KUKA KRL program: PPR_fullpath_2mm_split2.src

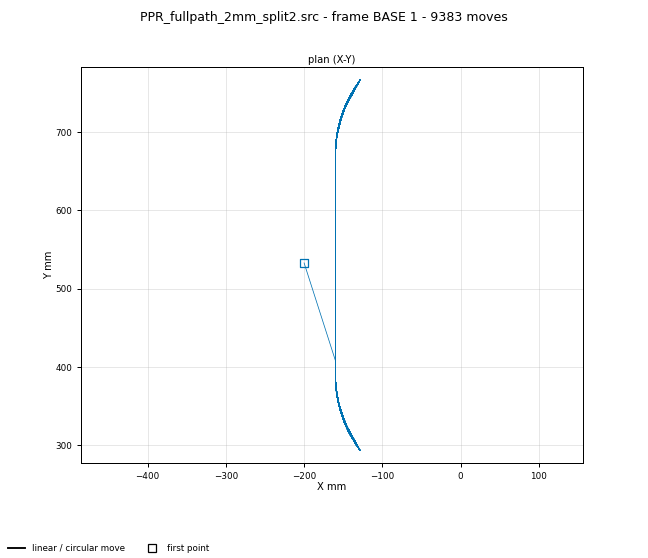
[picture p0: tool path of PPR_fullpath_2mm_split2.src in frame BASE 1, 9383 of 9384 moves have a stored position in this frame; points joined in program order, loops and branches not executed]
&ACCESS RVEO
&REL 11
&PARAM TEMPLATE = C:\KRC\Roboter\Template\vorgabe
&PARAM EDITMASK = *
DEF variable_helical2( )
;FOLD INI
  ;FOLD BASISTECH INI
    GLOBAL INTERRUPT DECL 3 WHEN $STOPMESS==TRUE DO IR_STOPM ( )
    INTERRUPT ON 3
    BAS (#INITMOV,0 )
  ;ENDFOLD (BASISTECH INI)
 ;FOLD USER INI


    ;Make your modifications here
  ;ENDFOLD (USER INI)
;ENDFOLD (INI)
ACTION(#AXIS_RESET,34,1000,#NOERROR,ERROR_CODE)
;FOLD PTP HOME  Vel= 100 % DEFAULT;%{PE}%MKUKATPBASIS,%CMOVE,%VPTP,%P 1:PTP, 2:HOME, 3:, 5:100, 7:DEFAULT
$BWDSTART = FALSE
PDAT_ACT=PDEFAULT
FDAT_ACT=FHOME
BAS (#PTP_PARAMS,100 )
$H_POS=XHOME
PTP  XHOME
;ENDFOLD
BAS(#TOOL,1)
BAS(#BASE,1)
$VEL_AXIS[1]=100
$VEL_AXIS[2]=100
$VEL_AXIS[3]=100
$VEL_AXIS[4]=100
$VEL_AXIS[5]=100
$VEL_AXIS[6]=100
$VEL_EXTAX[1]=100
$VEL_EXTAX[2]=100

$ACC_AXIS[1]=100
$ACC_AXIS[2]=100
$ACC_AXIS[3]=100
$ACC_AXIS[4]=100
$ACC_AXIS[5]=100
$ACC_AXIS[6]=100
$ACC_EXTAX[1]=100
$ACC_EXTAX[2]=100

SLIN {X  -200.000, Y  +533.000, Z    +0.000, A    +0.000, E1    +0.000, E3    +0.000, E4    +0.000}

SLIN {X  -160.000, Y  +408.284, Z    +0.000, E1   +56.435, E3  -372.434}
HALT
SPLINE
SPL {X  -160.000, Y  +395.668, Z    +0.000, E1   +56.446, E3  -354.661}
SPL {X  -159.894, Y  +382.991, Z    +0.000, E1   +56.419, E3  -336.663}
SPL {X  -159.213, Y  +372.948, Z    +0.000, E1   +56.290, E3  -321.768}
SPL {X  -158.141, Y  +364.480, Z    +0.000, E1   +56.110, E3  -308.694}
SPL {X  -156.499, Y  +355.511, Z    +0.000, E1   +55.854, E3  -294.378}
SPL {X  -154.489, Y  +347.168, Z    +0.000, E1   +55.487, E3  -280.503}
SPL {X  -152.108, Y  +339.170, Z    +0.000, E1   +55.085, E3  -266.814}
SPL {X  -149.149, Y  +330.880, Z    +0.000, E1   +54.560, E3  -252.178}
SPL {X  -146.188, Y  +323.769, Z    +0.000, E1   +53.991, E3  -239.222}
SPL {X  -143.516, Y  +318.068, Z    +0.000, E1   +53.476, E3  -228.622}
SPL {X  -140.415, Y  +312.095, Z    +0.000, E1   +52.896, E3  -217.355}
SPL {X  -128.706, Y  +293.749, Z    +0.000, E1   +44.636, E3  -115.294}
ENDSPLINE

SPLINE
SPL {X  -149.341, Y  +331.377, Z    +0.000, E1   +30.257, E3   -35.419}
SPL {X  -155.855, Y  +352.616, Z    +0.000, E1   +20.935, E3   -23.306}
SPL {X  -158.820, Y  +369.405, Z    +0.000, E1   +11.982, E3   -17.902}
SPL {X  -159.764, Y  +380.110, Z    +0.000, E1    +5.506, E3   -16.035}
SPL {X  -159.978, Y  +386.129, Z    +0.000, E1    +1.351, E3   -15.453}
SPL {X  -160.000, Y  +390.626, Z    +0.000, E1    -2.404, E3   -15.189}
SPL {X  -160.000, Y  +397.252, Z    +0.000, E1   -10.844, E3   -14.488}
SPL {X  -160.000, Y  +404.580, Z    +0.000, E1   -20.626, E3   -13.063}
SPL {X  -160.000, Y  +414.518, Z    +0.000, E1   -32.156, E3    -9.972}
SPL {X  -160.000, Y  +450.190, Z    +0.000, E1   -50.789, E3   +10.114}
SPL {X  -160.000, Y  +522.988, Z    +0.000, E1   -55.744, E3   +88.448}
SPL {X  -160.000, Y  +538.972, Z    +0.000, E1   -55.709, E3  +111.680}
SPL {X  -160.000, Y  +554.704, Z    +0.000, E1   -55.732, E3  +134.447}
SPL {X  -160.000, Y  +570.552, Z    +0.000, E1   -55.716, E3  +157.461}
SPL {X  -160.000, Y  +586.464, Z    +0.000, E1   -55.733, E3  +180.507}
SPL {X  -160.000, Y  +602.947, Z    +0.000, E1   -55.730, E3  +204.403}
SPL {X  -160.000, Y  +618.907, Z    +0.000, E1   -55.724, E3  +227.541}
SPL {X  -160.000, Y  +633.674, Z    +0.000, E1   -55.717, E3  +248.961}
SPL {X  -160.000, Y  +646.135, Z    +0.000, E1   -55.674, E3  +267.102}
SPL {X  -160.000, Y  +658.587, Z    +0.000, E1   -55.708, E3  +285.098}
SPL {X  -160.000, Y  +671.750, Z    +0.000, E1   -55.695, E3  +304.182}
SPL {X  -159.611, Y  +682.650, Z    +0.000, E1   -55.614, E3  +320.420}
SPL {X  -158.677, Y  +692.037, Z    +0.000, E1   -55.461, E3  +335.003}
SPL {X  -157.091, Y  +701.873, Z    +0.000, E1   -55.210, E3  +350.889}
SPL {X  -154.891, Y  +711.608, Z    +0.000, E1   -54.831, E3  +367.276}
SPL {X  -152.273, Y  +720.623, Z    +0.000, E1   -54.369, E3  +383.014}
SPL {X  -149.300, Y  +729.027, Z    +0.000, E1   -53.836, E3  +398.150}
SPL {X  -146.549, Y  +735.713, Z    +0.000, E1   -53.293, E3  +410.565}
SPL {X  -144.128, Y  +740.978, Z    +0.000, E1   -52.835, E3  +420.527}
SPL {X  -141.140, Y  +746.862, Z    +0.000, E1   -52.272, E3  +431.815}
SPL {X  -128.473, Y  +766.865, Z    +0.000, E1   -45.208, E3  +526.024}
ENDSPLINE

SPLINE
SPL {X  -149.609, Y  +728.220, Z    +0.000, E1   -30.103, E3  +611.717}
SPL {X  -157.346, Y  +700.520, Z    +0.000, E1   -17.449, E3  +626.438}
SPL {X  -159.391, Y  +685.442, Z    +0.000, E1    -8.940, E3  +630.323}
SPL {X  -159.974, Y  +674.384, Z    +0.000, E1    -1.914, E3  +631.675}
SPL {X  -160.000, Y  +668.854, Z    +0.000, E1    +3.008, E3  +632.026}
SPL {X  -160.000, Y  +662.175, Z    +0.000, E1   +11.518, E3  +632.797}
SPL {X  -160.000, Y  +654.447, Z    +0.000, E1   +21.734, E3  +634.422}
SPL {X  -160.000, Y  +641.600, Z    +0.000, E1   +35.681, E3  +638.687}
SPL {X  -160.000, Y  +601.361, Z    +0.000, E1   +52.744, E3  +662.649}
SPL {X  -160.000, Y  +531.662, Z    +0.000, E1   +56.951, E3  +734.638}
SPL {X  -160.000, Y  +513.172, Z    +0.000, E1   +56.969, E3  +760.194}
SPL {X  -160.000, Y  +498.160, Z    +0.000, E1   +56.531, E3  +783.807}
ENDSPLINE

SPLINE
SPL {X  -160.000, Y  +512.094, Z    +0.000, E1   +49.085, E3  +807.795}
ENDSPLINE

SPLINE
SPL {X  -160.000, Y  +491.347, Z    +0.000, E1   +50.960, E3  +833.461}
SPL {X  -160.000, Y  +470.538, Z    +0.000, E1   +52.629, E3  +858.147}
SPL {X  -160.000, Y  +453.213, Z    +0.000, E1   +53.894, E3  +877.585}
SPL {X  -160.000, Y  +440.734, Z    +0.000, E1   +54.729, E3  +891.367}
SPL {X  -160.000, Y  +423.596, Z    +0.000, E1   +55.911, E3  +909.259}
SPL {X  -160.000, Y  +408.178, Z    +0.000, E1   +56.432, E3  +927.720}
SPL {X  -160.000, Y  +395.668, Z    +0.000, E1   +56.446, E3  +945.336}
SPL {X  -159.894, Y  +382.991, Z    +0.000, E1   +56.419, E3  +963.334}
SPL {X  -159.213, Y  +372.948, Z    +0.000, E1   +56.290, E3  +978.228}
SPL {X  -158.141, Y  +364.480, Z    +0.000, E1   +56.110, E3  +991.303}
SPL {X  -156.499, Y  +355.511, Z    +0.000, E1   +55.854, E3 +1005.619}
SPL {X  -154.489, Y  +347.168, Z    +0.000, E1   +55.487, E3 +1019.493}
SPL {X  -152.108, Y  +339.170, Z    +0.000, E1   +55.085, E3 +1033.182}
SPL {X  -149.149, Y  +330.880, Z    +0.000, E1   +54.560, E3 +1047.818}
SPL {X  -146.188, Y  +323.769, Z    +0.000, E1   +53.991, E3 +1060.775}
SPL {X  -143.516, Y  +318.068, Z    +0.000, E1   +53.476, E3 +1071.374}
SPL {X  -140.415, Y  +312.095, Z    +0.000, E1   +52.896, E3 +1082.642}
SPL {X  -128.706, Y  +293.749, Z    +0.000, E1   +44.636, E3 +1184.702}
ENDSPLINE

SPLINE
SPL {X  -149.341, Y  +331.377, Z    +0.000, E1   +30.257, E3 +1264.578}
SPL {X  -155.855, Y  +352.616, Z    +0.000, E1   +20.935, E3 +1276.691}
SPL {X  -158.820, Y  +369.405, Z    +0.000, E1   +11.982, E3 +1282.094}
SPL {X  -159.764, Y  +380.110, Z    +0.000, E1    +5.506, E3 +1283.961}
SPL {X  -159.978, Y  +386.129, Z    +0.000, E1    +1.351, E3 +1284.543}
SPL {X  -160.000, Y  +390.626, Z    +0.000, E1    -2.404, E3 +1284.807}
SPL {X  -160.000, Y  +397.252, Z    +0.000, E1   -10.844, E3 +1285.508}
SPL {X  -160.000, Y  +404.580, Z    +0.000, E1   -20.626, E3 +1286.934}
SPL {X  -160.000, Y  +414.518, Z    +0.000, E1   -32.156, E3 +1290.024}
SPL {X  -160.000, Y  +450.190, Z    +0.000, E1   -50.789, E3 +1310.110}
SPL {X  -160.000, Y  +522.988, Z    +0.000, E1   -55.744, E3 +1388.444}
SPL {X  -160.000, Y  +538.972, Z    +0.000, E1   -55.709, E3 +1411.677}
SPL {X  -160.000, Y  +554.704, Z    +0.000, E1   -55.732, E3 +1434.443}
SPL {X  -160.000, Y  +570.552, Z    +0.000, E1   -55.716, E3 +1457.458}
SPL {X  -160.000, Y  +586.464, Z    +0.000, E1   -55.733, E3 +1480.503}
SPL {X  -160.000, Y  +602.947, Z    +0.000, E1   -55.730, E3 +1504.400}
SPL {X  -160.000, Y  +618.907, Z    +0.000, E1   -55.724, E3 +1527.537}
SPL {X  -160.000, Y  +633.674, Z    +0.000, E1   -55.717, E3 +1548.957}
SPL {X  -160.000, Y  +646.135, Z    +0.000, E1   -55.674, E3 +1567.098}
SPL {X  -160.000, Y  +658.587, Z    +0.000, E1   -55.708, E3 +1585.094}
SPL {X  -160.000, Y  +671.750, Z    +0.000, E1   -55.695, E3 +1604.179}
SPL {X  -159.611, Y  +682.650, Z    +0.000, E1   -55.614, E3 +1620.417}
SPL {X  -158.677, Y  +692.037, Z    +0.000, E1   -55.461, E3 +1635.000}
SPL {X  -157.091, Y  +701.873, Z    +0.000, E1   -55.210, E3 +1650.886}
SPL {X  -154.891, Y  +711.608, Z    +0.000, E1   -54.831, E3 +1667.273}
SPL {X  -152.273, Y  +720.623, Z    +0.000, E1   -54.369, E3 +1683.010}
SPL {X  -149.300, Y  +729.027, Z    +0.000, E1   -53.836, E3 +1698.146}
SPL {X  -146.549, Y  +735.713, Z    +0.000, E1   -53.293, E3 +1710.561}
SPL {X  -144.128, Y  +740.978, Z    +0.000, E1   -52.835, E3 +1720.524}
SPL {X  -141.140, Y  +746.862, Z    +0.000, E1   -52.272, E3 +1731.811}
SPL {X  -128.473, Y  +766.865, Z    +0.000, E1   -45.208, E3 +1826.021}
ENDSPLINE

SPLINE
SPL {X  -149.609, Y  +728.220, Z    +0.000, E1   -30.103, E3 +1911.713}
SPL {X  -157.346, Y  +700.520, Z    +0.000, E1   -17.449, E3 +1926.434}
SPL {X  -159.391, Y  +685.442, Z    +0.000, E1    -8.940, E3 +1930.319}
SPL {X  -159.974, Y  +674.384, Z    +0.000, E1    -1.914, E3 +1931.671}
SPL {X  -160.000, Y  +668.854, Z    +0.000, E1    +3.008, E3 +1932.022}
SPL {X  -160.000, Y  +662.175, Z    +0.000, E1   +11.518, E3 +1932.793}
SPL {X  -160.000, Y  +654.447, Z    +0.000, E1   +21.734, E3 +1934.419}
SPL {X  -160.000, Y  +641.600, Z    +0.000, E1   +35.681, E3 +1938.684}
SPL {X  -160.000, Y  +601.361, Z    +0.000, E1   +52.744, E3 +1962.645}
SPL {X  -160.000, Y  +531.662, Z    +0.000, E1   +56.951, E3 +2034.635}
SPL {X  -160.000, Y  +513.172, Z    +0.000, E1   +56.969, E3 +2060.190}
SPL {X  -160.000, Y  +498.160, Z    +0.000, E1   +56.531, E3 +2083.803}
ENDSPLINE

SPLINE
SPL {X  -160.000, Y  +512.094, Z    +0.000, E1   +49.085, E3 +2107.791}
ENDSPLINE

SPLINE
SPL {X  -160.000, Y  +491.347, Z    +0.000, E1   +50.960, E3 +2133.458}
SPL {X  -160.000, Y  +470.538, Z    +0.000, E1   +52.629, E3 +2158.144}
SPL {X  -160.000, Y  +453.213, Z    +0.000, E1   +53.894, E3 +2177.582}
SPL {X  -160.000, Y  +440.734, Z    +0.000, E1   +54.729, E3 +2191.364}
SPL {X  -160.000, Y  +423.596, Z    +0.000, E1   +55.911, E3 +2209.256}
SPL {X  -160.000, Y  +408.178, Z    +0.000, E1   +56.432, E3 +2227.717}
SPL {X  -160.000, Y  +395.668, Z    +0.000, E1   +56.446, E3 +2245.332}
SPL {X  -159.894, Y  +382.991, Z    +0.000, E1   +56.419, E3 +2263.330}
SPL {X  -159.213, Y  +372.948, Z    +0.000, E1   +56.290, E3 +2278.225}
SPL {X  -158.141, Y  +364.480, Z    +0.000, E1   +56.110, E3 +2291.299}
SPL {X  -156.499, Y  +355.511, Z    +0.000, E1   +55.854, E3 +2305.615}
SPL {X  -154.489, Y  +347.168, Z    +0.000, E1   +55.487, E3 +2319.490}
SPL {X  -152.108, Y  +339.170, Z    +0.000, E1   +55.085, E3 +2333.179}
SPL {X  -149.149, Y  +330.880, Z    +0.000, E1   +54.560, E3 +2347.814}
SPL {X  -146.188, Y  +323.769, Z    +0.000, E1   +53.991, E3 +2360.771}
SPL {X  -143.516, Y  +318.068, Z    +0.000, E1   +53.476, E3 +2371.371}
SPL {X  -140.415, Y  +312.095, Z    +0.000, E1   +52.896, E3 +2382.638}
SPL {X  -128.706, Y  +293.749, Z    +0.000, E1   +44.636, E3 +2484.699}
ENDSPLINE

SPLINE
SPL {X  -149.341, Y  +331.377, Z    +0.000, E1   +30.257, E3 +2564.574}
SPL {X  -155.855, Y  +352.616, Z    +0.000, E1   +20.935, E3 +2576.687}
SPL {X  -158.820, Y  +369.405, Z    +0.000, E1   +11.982, E3 +2582.091}
SPL {X  -159.764, Y  +380.110, Z    +0.000, E1    +5.506, E3 +2583.957}
SPL {X  -159.978, Y  +386.129, Z    +0.000, E1    +1.351, E3 +2584.540}
SPL {X  -160.000, Y  +390.626, Z    +0.000, E1    -2.404, E3 +2584.804}
SPL {X  -160.000, Y  +397.252, Z    +0.000, E1   -10.844, E3 +2585.504}
SPL {X  -160.000, Y  +404.580, Z    +0.000, E1   -20.626, E3 +2586.930}
SPL {X  -160.000, Y  +414.518, Z    +0.000, E1   -32.156, E3 +2590.021}
SPL {X  -160.000, Y  +450.190, Z    +0.000, E1   -50.789, E3 +2610.106}
SPL {X  -160.000, Y  +522.988, Z    +0.000, E1   -55.744, E3 +2688.441}
SPL {X  -160.000, Y  +538.972, Z    +0.000, E1   -55.709, E3 +2711.673}
SPL {X  -160.000, Y  +554.704, Z    +0.000, E1   -55.732, E3 +2734.439}
SPL {X  -160.000, Y  +570.552, Z    +0.000, E1   -55.716, E3 +2757.454}
SPL {X  -160.000, Y  +586.464, Z    +0.000, E1   -55.733, E3 +2780.499}
SPL {X  -160.000, Y  +602.947, Z    +0.000, E1   -55.730, E3 +2804.396}
SPL {X  -160.000, Y  +618.907, Z    +0.000, E1   -55.724, E3 +2827.534}
SPL {X  -160.000, Y  +633.674, Z    +0.000, E1   -55.717, E3 +2848.954}
SPL {X  -160.000, Y  +646.135, Z    +0.000, E1   -55.674, E3 +2867.094}
SPL {X  -160.000, Y  +658.587, Z    +0.000, E1   -55.708, E3 +2885.090}
SPL {X  -160.000, Y  +671.750, Z    +0.000, E1   -55.695, E3 +2904.175}
SPL {X  -159.611, Y  +682.650, Z    +0.000, E1   -55.614, E3 +2920.413}
SPL {X  -158.677, Y  +692.037, Z    +0.000, E1   -55.461, E3 +2934.996}
SPL {X  -157.091, Y  +701.873, Z    +0.000, E1   -55.210, E3 +2950.882}
SPL {X  -154.891, Y  +711.608, Z    +0.000, E1   -54.831, E3 +2967.269}
SPL {X  -152.273, Y  +720.623, Z    +0.000, E1   -54.369, E3 +2983.007}
SPL {X  -149.300, Y  +729.027, Z    +0.000, E1   -53.836, E3 +2998.143}
SPL {X  -146.549, Y  +735.713, Z    +0.000, E1   -53.293, E3 +3010.557}
SPL {X  -144.128, Y  +740.978, Z    +0.000, E1   -52.835, E3 +3020.520}
SPL {X  -141.140, Y  +746.862, Z    +0.000, E1   -52.272, E3 +3031.808}
SPL {X  -128.473, Y  +766.865, Z    +0.000, E1   -45.208, E3 +3126.017}
ENDSPLINE

SPLINE
SPL {X  -149.609, Y  +728.220, Z    +0.000, E1   -30.103, E3 +3211.710}
SPL {X  -157.346, Y  +700.520, Z    +0.000, E1   -17.449, E3 +3226.431}
SPL {X  -159.391, Y  +685.442, Z    +0.000, E1    -8.940, E3 +3230.316}
SPL {X  -159.974, Y  +674.384, Z    +0.000, E1    -1.914, E3 +3231.668}
SPL {X  -160.000, Y  +668.854, Z    +0.000, E1    +3.008, E3 +3232.019}
SPL {X  -160.000, Y  +662.175, Z    +0.000, E1   +11.518, E3 +3232.789}
SPL {X  -160.000, Y  +654.447, Z    +0.000, E1   +21.734, E3 +3234.415}
SPL {X  -160.000, Y  +641.600, Z    +0.000, E1   +35.681, E3 +3238.680}
SPL {X  -160.000, Y  +601.361, Z    +0.000, E1   +52.744, E3 +3262.642}
SPL {X  -160.000, Y  +531.662, Z    +0.000, E1   +56.951, E3 +3334.631}
SPL {X  -160.000, Y  +513.172, Z    +0.000, E1   +56.969, E3 +3360.187}
SPL {X  -160.000, Y  +498.160, Z    +0.000, E1   +56.531, E3 +3383.800}
ENDSPLINE

SPLINE
SPL {X  -160.000, Y  +512.094, Z    +0.000, E1   +49.085, E3 +3407.787}
ENDSPLINE

SPLINE
SPL {X  -160.000, Y  +491.347, Z    +0.000, E1   +50.960, E3 +3433.454}
SPL {X  -160.000, Y  +470.538, Z    +0.000, E1   +52.629, E3 +3458.140}
SPL {X  -160.000, Y  +453.213, Z    +0.000, E1   +53.894, E3 +3477.578}
SPL {X  -160.000, Y  +440.734, Z    +0.000, E1   +54.729, E3 +3491.360}
SPL {X  -160.000, Y  +423.596, Z    +0.000, E1   +55.911, E3 +3509.252}
SPL {X  -160.000, Y  +408.178, Z    +0.000, E1   +56.432, E3 +3527.713}
SPL {X  -160.000, Y  +395.668, Z    +0.000, E1   +56.446, E3 +3545.328}
SPL {X  -159.894, Y  +382.991, Z    +0.000, E1   +56.419, E3 +3563.326}
SPL {X  -159.213, Y  +372.948, Z    +0.000, E1   +56.290, E3 +3578.221}
SPL {X  -158.141, Y  +364.480, Z    +0.000, E1   +56.110, E3 +3591.295}
SPL {X  -156.499, Y  +355.511, Z    +0.000, E1   +55.854, E3 +3605.611}
SPL {X  -154.489, Y  +347.168, Z    +0.000, E1   +55.487, E3 +3619.486}
SPL {X  -152.108, Y  +339.170, Z    +0.000, E1   +55.085, E3 +3633.175}
SPL {X  -149.149, Y  +330.880, Z    +0.000, E1   +54.560, E3 +3647.811}
SPL {X  -146.188, Y  +323.769, Z    +0.000, E1   +53.991, E3 +3660.767}
SPL {X  -143.516, Y  +318.068, Z    +0.000, E1   +53.476, E3 +3671.367}
SPL {X  -140.415, Y  +312.095, Z    +0.000, E1   +52.896, E3 +3682.634}
SPL {X  -128.706, Y  +293.749, Z    +0.000, E1   +44.636, E3 +3784.695}
ENDSPLINE

SPLINE
SPL {X  -149.341, Y  +331.377, Z    +0.000, E1   +30.257, E3 +3864.571}
SPL {X  -155.855, Y  +352.616, Z    +0.000, E1   +20.935, E3 +3876.683}
SPL {X  -158.820, Y  +369.405, Z    +0.000, E1   +11.982, E3 +3882.087}
SPL {X  -159.764, Y  +380.110, Z    +0.000, E1    +5.506, E3 +3883.954}
SPL {X  -159.978, Y  +386.129, Z    +0.000, E1    +1.351, E3 +3884.536}
SPL {X  -160.000, Y  +390.626, Z    +0.000, E1    -2.404, E3 +3884.800}
SPL {X  -160.000, Y  +397.252, Z    +0.000, E1   -10.844, E3 +3885.501}
SPL {X  -160.000, Y  +404.580, Z    +0.000, E1   -20.626, E3 +3886.926}
SPL {X  -160.000, Y  +414.518, Z    +0.000, E1   -32.156, E3 +3890.017}
SPL {X  -160.000, Y  +450.190, Z    +0.000, E1   -50.789, E3 +3910.103}
SPL {X  -160.000, Y  +522.988, Z    +0.000, E1   -55.744, E3 +3988.437}
SPL {X  -160.000, Y  +538.972, Z    +0.000, E1   -55.709, E3 +4011.669}
SPL {X  -160.000, Y  +554.704, Z    +0.000, E1   -55.732, E3 +4034.436}
SPL {X  -160.000, Y  +570.552, Z    +0.000, E1   -55.716, E3 +4057.450}
SPL {X  -160.000, Y  +586.464, Z    +0.000, E1   -55.733, E3 +4080.496}
SPL {X  -160.000, Y  +602.947, Z    +0.000, E1   -55.730, E3 +4104.392}
SPL {X  -160.000, Y  +618.907, Z    +0.000, E1   -55.724, E3 +4127.530}
SPL {X  -160.000, Y  +633.674, Z    +0.000, E1   -55.717, E3 +4148.950}
SPL {X  -160.000, Y  +646.135, Z    +0.000, E1   -55.674, E3 +4167.091}
SPL {X  -160.000, Y  +658.587, Z    +0.000, E1   -55.708, E3 +4185.087}
SPL {X  -160.000, Y  +671.750, Z    +0.000, E1   -55.695, E3 +4204.172}
SPL {X  -159.611, Y  +682.650, Z    +0.000, E1   -55.614, E3 +4220.409}
SPL {X  -158.677, Y  +692.037, Z    +0.000, E1   -55.461, E3 +4234.992}
SPL {X  -157.091, Y  +701.873, Z    +0.000, E1   -55.210, E3 +4250.879}
SPL {X  -154.891, Y  +711.608, Z    +0.000, E1   -54.831, E3 +4267.265}
SPL {X  -152.273, Y  +720.623, Z    +0.000, E1   -54.369, E3 +4283.003}
SPL {X  -149.300, Y  +729.027, Z    +0.000, E1   -53.836, E3 +4298.139}
SPL {X  -146.549, Y  +735.713, Z    +0.000, E1   -53.293, E3 +4310.554}
SPL {X  -144.128, Y  +740.978, Z    +0.000, E1   -52.835, E3 +4320.516}
SPL {X  -141.140, Y  +746.862, Z    +0.000, E1   -52.272, E3 +4331.804}
SPL {X  -128.473, Y  +766.865, Z    +0.000, E1   -45.208, E3 +4426.013}
ENDSPLINE

SPLINE
SPL {X  -149.609, Y  +728.220, Z    +0.000, E1   -30.103, E3 +4511.706}
SPL {X  -157.346, Y  +700.520, Z    +0.000, E1   -17.449, E3 +4526.427}
SPL {X  -159.391, Y  +685.442, Z    +0.000, E1    -8.940, E3 +4530.312}
SPL {X  -159.974, Y  +674.384, Z    +0.000, E1    -1.914, E3 +4531.664}
SPL {X  -160.000, Y  +668.854, Z    +0.000, E1    +3.008, E3 +4532.015}
SPL {X  -160.000, Y  +662.175, Z    +0.000, E1   +11.518, E3 +4532.786}
SPL {X  -160.000, Y  +654.447, Z    +0.000, E1   +21.734, E3 +4534.411}
SPL {X  -160.000, Y  +641.600, Z    +0.000, E1   +35.681, E3 +4538.676}
SPL {X  -160.000, Y  +601.361, Z    +0.000, E1   +52.744, E3 +4562.638}
SPL {X  -160.000, Y  +531.662, Z    +0.000, E1   +56.951, E3 +4634.627}
SPL {X  -160.000, Y  +513.172, Z    +0.000, E1   +56.969, E3 +4660.183}
SPL {X  -160.000, Y  +498.160, Z    +0.000, E1   +56.531, E3 +4683.796}
ENDSPLINE

SPLINE
SPL {X  -160.000, Y  +512.094, Z    +0.000, E1   +49.085, E3 +4707.784}
ENDSPLINE

SPLINE
SPL {X  -160.000, Y  +491.347, Z    +0.000, E1   +50.960, E3 +4733.450}
SPL {X  -160.000, Y  +470.538, Z    +0.000, E1   +52.629, E3 +4758.136}
SPL {X  -160.000, Y  +453.213, Z    +0.000, E1   +53.894, E3 +4777.574}
SPL {X  -160.000, Y  +440.734, Z    +0.000, E1   +54.729, E3 +4791.356}
SPL {X  -160.000, Y  +423.596, Z    +0.000, E1   +55.911, E3 +4809.248}
SPL {X  -160.000, Y  +408.178, Z    +0.000, E1   +56.432, E3 +4827.709}
SPL {X  -160.000, Y  +395.668, Z    +0.000, E1   +56.446, E3 +4845.325}
SPL {X  -159.894, Y  +382.991, Z    +0.000, E1   +56.419, E3 +4863.323}
SPL {X  -159.213, Y  +372.948, Z    +0.000, E1   +56.290, E3 +4878.217}
SPL {X  -158.141, Y  +364.480, Z    +0.000, E1   +56.110, E3 +4891.292}
SPL {X  -156.499, Y  +355.511, Z    +0.000, E1   +55.854, E3 +4905.608}
SPL {X  -154.489, Y  +347.168, Z    +0.000, E1   +55.487, E3 +4919.482}
SPL {X  -152.108, Y  +339.170, Z    +0.000, E1   +55.085, E3 +4933.172}
SPL {X  -149.149, Y  +330.880, Z    +0.000, E1   +54.560, E3 +4947.807}
SPL {X  -146.188, Y  +323.769, Z    +0.000, E1   +53.991, E3 +4960.764}
SPL {X  -143.516, Y  +318.068, Z    +0.000, E1   +53.476, E3 +4971.363}
SPL {X  -140.415, Y  +312.095, Z    +0.000, E1   +52.896, E3 +4982.631}
SPL {X  -128.706, Y  +293.749, Z    +0.000, E1   +44.636, E3 +5084.691}
ENDSPLINE

SPLINE
SPL {X  -149.341, Y  +331.377, Z    +0.000, E1   +30.257, E3 +5164.567}
SPL {X  -155.855, Y  +352.616, Z    +0.000, E1   +20.935, E3 +5176.680}
SPL {X  -158.820, Y  +369.405, Z    +0.000, E1   +11.982, E3 +5182.084}
SPL {X  -159.764, Y  +380.110, Z    +0.000, E1    +5.506, E3 +5183.950}
SPL {X  -159.978, Y  +386.129, Z    +0.000, E1    +1.351, E3 +5184.532}
SPL {X  -160.000, Y  +390.626, Z    +0.000, E1    -2.404, E3 +5184.796}
SPL {X  -160.000, Y  +397.252, Z    +0.000, E1   -10.844, E3 +5185.497}
SPL {X  -160.000, Y  +404.580, Z    +0.000, E1   -20.626, E3 +5186.923}
SPL {X  -160.000, Y  +414.518, Z    +0.000, E1   -32.156, E3 +5190.013}
SPL {X  -160.000, Y  +450.190, Z    +0.000, E1   -50.789, E3 +5210.099}
SPL {X  -160.000, Y  +522.988, Z    +0.000, E1   -55.744, E3 +5288.433}
SPL {X  -160.000, Y  +538.972, Z    +0.000, E1   -55.709, E3 +5311.666}
SPL {X  -160.000, Y  +554.704, Z    +0.000, E1   -55.732, E3 +5334.432}
SPL {X  -160.000, Y  +570.552, Z    +0.000, E1   -55.716, E3 +5357.447}
SPL {X  -160.000, Y  +586.464, Z    +0.000, E1   -55.733, E3 +5380.492}
SPL {X  -160.000, Y  +602.947, Z    +0.000, E1   -55.730, E3 +5404.389}
SPL {X  -160.000, Y  +618.907, Z    +0.000, E1   -55.724, E3 +5427.527}
SPL {X  -160.000, Y  +633.674, Z    +0.000, E1   -55.717, E3 +5448.947}
SPL {X  -160.000, Y  +646.135, Z    +0.000, E1   -55.674, E3 +5467.087}
SPL {X  -160.000, Y  +658.587, Z    +0.000, E1   -55.708, E3 +5485.083}
SPL {X  -160.000, Y  +671.750, Z    +0.000, E1   -55.695, E3 +5504.168}
SPL {X  -159.611, Y  +682.650, Z    +0.000, E1   -55.614, E3 +5520.406}
SPL {X  -158.677, Y  +692.037, Z    +0.000, E1   -55.461, E3 +5534.989}
SPL {X  -157.091, Y  +701.873, Z    +0.000, E1   -55.210, E3 +5550.875}
SPL {X  -154.891, Y  +711.608, Z    +0.000, E1   -54.831, E3 +5567.262}
SPL {X  -152.273, Y  +720.623, Z    +0.000, E1   -54.369, E3 +5582.999}
SPL {X  -149.300, Y  +729.027, Z    +0.000, E1   -53.836, E3 +5598.135}
SPL {X  -146.549, Y  +735.713, Z    +0.000, E1   -53.293, E3 +5610.550}
SPL {X  -144.128, Y  +740.978, Z    +0.000, E1   -52.835, E3 +5620.513}
SPL {X  -141.140, Y  +746.862, Z    +0.000, E1   -52.272, E3 +5631.800}
SPL {X  -128.473, Y  +766.865, Z    +0.000, E1   -45.208, E3 +5726.010}
ENDSPLINE

SPLINE
SPL {X  -149.609, Y  +728.220, Z    +0.000, E1   -30.103, E3 +5811.703}
SPL {X  -157.346, Y  +700.520, Z    +0.000, E1   -17.449, E3 +5826.423}
SPL {X  -159.391, Y  +685.442, Z    +0.000, E1    -8.940, E3 +5830.309}
SPL {X  -159.974, Y  +674.384, Z    +0.000, E1    -1.914, E3 +5831.660}
SPL {X  -160.000, Y  +668.854, Z    +0.000, E1    +3.008, E3 +5832.011}
SPL {X  -160.000, Y  +662.175, Z    +0.000, E1   +11.518, E3 +5832.782}
SPL {X  -160.000, Y  +654.447, Z    +0.000, E1   +21.734, E3 +5834.408}
SPL {X  -160.000, Y  +641.600, Z    +0.000, E1   +35.681, E3 +5838.673}
SPL {X  -160.000, Y  +601.361, Z    +0.000, E1   +52.744, E3 +5862.635}
SPL {X  -160.000, Y  +531.662, Z    +0.000, E1   +56.951, E3 +5934.624}
SPL {X  -160.000, Y  +513.172, Z    +0.000, E1   +56.969, E3 +5960.179}
SPL {X  -160.000, Y  +498.160, Z    +0.000, E1   +56.531, E3 +5983.792}
ENDSPLINE

SPLINE
SPL {X  -160.000, Y  +512.094, Z    +0.000, E1   +49.085, E3 +6007.780}
ENDSPLINE

SPLINE
SPL {X  -160.000, Y  +491.347, Z    +0.000, E1   +50.960, E3 +6033.447}
SPL {X  -160.000, Y  +470.538, Z    +0.000, E1   +52.629, E3 +6058.133}
SPL {X  -160.000, Y  +453.213, Z    +0.000, E1   +53.894, E3 +6077.571}
SPL {X  -160.000, Y  +440.734, Z    +0.000, E1   +54.729, E3 +6091.353}
SPL {X  -160.000, Y  +423.596, Z    +0.000, E1   +55.911, E3 +6109.245}
SPL {X  -160.000, Y  +408.178, Z    +0.000, E1   +56.432, E3 +6127.706}
SPL {X  -160.000, Y  +395.668, Z    +0.000, E1   +56.446, E3 +6145.321}
SPL {X  -159.894, Y  +382.991, Z    +0.000, E1   +56.419, E3 +6163.319}
SPL {X  -159.213, Y  +372.948, Z    +0.000, E1   +56.290, E3 +6178.214}
SPL {X  -158.141, Y  +364.480, Z    +0.000, E1   +56.110, E3 +6191.288}
SPL {X  -156.499, Y  +355.511, Z    +0.000, E1   +55.854, E3 +6205.604}
SPL {X  -154.489, Y  +347.168, Z    +0.000, E1   +55.487, E3 +6219.479}
SPL {X  -152.108, Y  +339.170, Z    +0.000, E1   +55.085, E3 +6233.168}
SPL {X  -149.149, Y  +330.880, Z    +0.000, E1   +54.560, E3 +6247.804}
SPL {X  -146.188, Y  +323.769, Z    +0.000, E1   +53.991, E3 +6260.760}
SPL {X  -143.516, Y  +318.068, Z    +0.000, E1   +53.476, E3 +6271.360}
SPL {X  -140.415, Y  +312.095, Z    +0.000, E1   +52.896, E3 +6282.627}
SPL {X  -128.706, Y  +293.749, Z    +0.000, E1   +44.636, E3 +6384.688}
ENDSPLINE

SPLINE
SPL {X  -149.341, Y  +331.377, Z    +0.000, E1   +30.257, E3 +6464.563}
SPL {X  -155.855, Y  +352.616, Z    +0.000, E1   +20.935, E3 +6476.676}
SPL {X  -158.820, Y  +369.405, Z    +0.000, E1   +11.982, E3 +6482.080}
SPL {X  -159.764, Y  +380.110, Z    +0.000, E1    +5.506, E3 +6483.946}
SPL {X  -159.978, Y  +386.129, Z    +0.000, E1    +1.351, E3 +6484.529}
SPL {X  -160.000, Y  +390.626, Z    +0.000, E1    -2.404, E3 +6484.793}
SPL {X  -160.000, Y  +397.252, Z    +0.000, E1   -10.844, E3 +6485.494}
SPL {X  -160.000, Y  +404.580, Z    +0.000, E1   -20.626, E3 +6486.919}
SPL {X  -160.000, Y  +414.518, Z    +0.000, E1   -32.156, E3 +6490.010}
SPL {X  -160.000, Y  +450.190, Z    +0.000, E1   -50.789, E3 +6510.096}
SPL {X  -160.000, Y  +522.988, Z    +0.000, E1   -55.744, E3 +6588.430}
SPL {X  -160.000, Y  +538.972, Z    +0.000, E1   -55.709, E3 +6611.662}
SPL {X  -160.000, Y  +554.704, Z    +0.000, E1   -55.732, E3 +6634.428}
SPL {X  -160.000, Y  +570.552, Z    +0.000, E1   -55.716, E3 +6657.443}
SPL {X  -160.000, Y  +586.464, Z    +0.000, E1   -55.733, E3 +6680.488}
SPL {X  -160.000, Y  +602.947, Z    +0.000, E1   -55.730, E3 +6704.385}
SPL {X  -160.000, Y  +618.907, Z    +0.000, E1   -55.724, E3 +6727.523}
SPL {X  -160.000, Y  +633.674, Z    +0.000, E1   -55.717, E3 +6748.943}
SPL {X  -160.000, Y  +646.135, Z    +0.000, E1   -55.674, E3 +6767.083}
SPL {X  -160.000, Y  +658.587, Z    +0.000, E1   -55.708, E3 +6785.079}
SPL {X  -160.000, Y  +671.750, Z    +0.000, E1   -55.695, E3 +6804.164}
SPL {X  -159.611, Y  +682.650, Z    +0.000, E1   -55.614, E3 +6820.402}
SPL {X  -158.677, Y  +692.037, Z    +0.000, E1   -55.461, E3 +6834.985}
SPL {X  -157.091, Y  +701.873, Z    +0.000, E1   -55.210, E3 +6850.871}
SPL {X  -154.891, Y  +711.608, Z    +0.000, E1   -54.831, E3 +6867.258}
SPL {X  -152.273, Y  +720.623, Z    +0.000, E1   -54.369, E3 +6882.996}
SPL {X  -149.300, Y  +729.027, Z    +0.000, E1   -53.836, E3 +6898.132}
SPL {X  -146.549, Y  +735.713, Z    +0.000, E1   -53.293, E3 +6910.546}
SPL {X  -144.128, Y  +740.978, Z    +0.000, E1   -52.835, E3 +6920.509}
SPL {X  -141.140, Y  +746.862, Z    +0.000, E1   -52.272, E3 +6931.797}
SPL {X  -128.473, Y  +766.865, Z    +0.000, E1   -45.208, E3 +7026.006}
ENDSPLINE

SPLINE
SPL {X  -149.609, Y  +728.220, Z    +0.000, E1   -30.103, E3 +7111.699}
SPL {X  -157.346, Y  +700.520, Z    +0.000, E1   -17.449, E3 +7126.420}
SPL {X  -159.391, Y  +685.442, Z    +0.000, E1    -8.940, E3 +7130.305}
SPL {X  -159.974, Y  +674.384, Z    +0.000, E1    -1.914, E3 +7131.657}
SPL {X  -160.000, Y  +668.854, Z    +0.000, E1    +3.008, E3 +7132.008}
SPL {X  -160.000, Y  +662.175, Z    +0.000, E1   +11.518, E3 +7132.778}
SPL {X  -160.000, Y  +654.447, Z    +0.000, E1   +21.734, E3 +7134.404}
SPL {X  -160.000, Y  +641.600, Z    +0.000, E1   +35.681, E3 +7138.669}
SPL {X  -160.000, Y  +601.361, Z    +0.000, E1   +52.744, E3 +7162.631}
SPL {X  -160.000, Y  +531.662, Z    +0.000, E1   +56.951, E3 +7234.620}
SPL {X  -160.000, Y  +513.172, Z    +0.000, E1   +56.969, E3 +7260.176}
SPL {X  -160.000, Y  +498.160, Z    +0.000, E1   +56.531, E3 +7283.789}
ENDSPLINE

SPLINE
SPL {X  -160.000, Y  +512.094, Z    +0.000, E1   +49.085, E3 +7307.777}
ENDSPLINE

SPLINE
SPL {X  -160.000, Y  +491.347, Z    +0.000, E1   +50.960, E3 +7333.443}
SPL {X  -160.000, Y  +470.538, Z    +0.000, E1   +52.629, E3 +7358.129}
SPL {X  -160.000, Y  +453.213, Z    +0.000, E1   +53.894, E3 +7377.567}
SPL {X  -160.000, Y  +440.734, Z    +0.000, E1   +54.729, E3 +7391.349}
SPL {X  -160.000, Y  +423.596, Z    +0.000, E1   +55.911, E3 +7409.241}
SPL {X  -160.000, Y  +408.178, Z    +0.000, E1   +56.432, E3 +7427.702}
SPL {X  -160.000, Y  +395.668, Z    +0.000, E1   +56.446, E3 +7445.317}
SPL {X  -159.894, Y  +382.991, Z    +0.000, E1   +56.419, E3 +7463.316}
SPL {X  -159.213, Y  +372.948, Z    +0.000, E1   +56.290, E3 +7478.210}
SPL {X  -158.141, Y  +364.480, Z    +0.000, E1   +56.110, E3 +7491.284}
SPL {X  -156.499, Y  +355.511, Z    +0.000, E1   +55.854, E3 +7505.601}
SPL {X  -154.489, Y  +347.168, Z    +0.000, E1   +55.487, E3 +7519.475}
SPL {X  -152.108, Y  +339.170, Z    +0.000, E1   +55.085, E3 +7533.164}
SPL {X  -149.149, Y  +330.880, Z    +0.000, E1   +54.560, E3 +7547.800}
SPL {X  -146.188, Y  +323.769, Z    +0.000, E1   +53.991, E3 +7560.757}
SPL {X  -143.516, Y  +318.068, Z    +0.000, E1   +53.476, E3 +7571.356}
SPL {X  -140.415, Y  +312.095, Z    +0.000, E1   +52.896, E3 +7582.624}
SPL {X  -128.706, Y  +293.749, Z    +0.000, E1   +44.636, E3 +7684.684}
ENDSPLINE

SPLINE
SPL {X  -149.341, Y  +331.377, Z    +0.000, E1   +30.257, E3 +7764.560}
SPL {X  -155.855, Y  +352.616, Z    +0.000, E1   +20.935, E3 +7776.673}
SPL {X  -158.820, Y  +369.405, Z    +0.000, E1   +11.982, E3 +7782.076}
SPL {X  -159.764, Y  +380.110, Z    +0.000, E1    +5.506, E3 +7783.943}
SPL {X  -159.978, Y  +386.129, Z    +0.000, E1    +1.351, E3 +7784.525}
SPL {X  -160.000, Y  +390.626, Z    +0.000, E1    -2.404, E3 +7784.789}
SPL {X  -160.000, Y  +397.252, Z    +0.000, E1   -10.844, E3 +7785.490}
SPL {X  -160.000, Y  +404.580, Z    +0.000, E1   -20.626, E3 +7786.916}
SPL {X  -160.000, Y  +414.518, Z    +0.000, E1   -32.156, E3 +7790.006}
SPL {X  -160.000, Y  +450.190, Z    +0.000, E1   -50.789, E3 +7810.092}
SPL {X  -160.000, Y  +522.988, Z    +0.000, E1   -55.744, E3 +7888.426}
SPL {X  -160.000, Y  +538.972, Z    +0.000, E1   -55.709, E3 +7911.658}
SPL {X  -160.000, Y  +554.704, Z    +0.000, E1   -55.732, E3 +7934.425}
SPL {X  -160.000, Y  +570.552, Z    +0.000, E1   -55.716, E3 +7957.440}
SPL {X  -160.000, Y  +586.464, Z    +0.000, E1   -55.733, E3 +7980.485}
SPL {X  -160.000, Y  +602.947, Z    +0.000, E1   -55.730, E3 +8004.381}
SPL {X  -160.000, Y  +618.907, Z    +0.000, E1   -55.724, E3 +8027.519}
SPL {X  -160.000, Y  +633.674, Z    +0.000, E1   -55.717, E3 +8048.939}
SPL {X  -160.000, Y  +646.135, Z    +0.000, E1   -55.674, E3 +8067.080}
SPL {X  -160.000, Y  +658.587, Z    +0.000, E1   -55.708, E3 +8085.076}
SPL {X  -160.000, Y  +671.750, Z    +0.000, E1   -55.695, E3 +8104.161}
SPL {X  -159.611, Y  +682.650, Z    +0.000, E1   -55.614, E3 +8120.399}
SPL {X  -158.677, Y  +692.037, Z    +0.000, E1   -55.461, E3 +8134.982}
SPL {X  -157.091, Y  +701.873, Z    +0.000, E1   -55.210, E3 +8150.868}
SPL {X  -154.891, Y  +711.608, Z    +0.000, E1   -54.831, E3 +8167.255}
SPL {X  -152.273, Y  +720.623, Z    +0.000, E1   -54.369, E3 +8182.992}
SPL {X  -149.300, Y  +729.027, Z    +0.000, E1   -53.836, E3 +8198.128}
SPL {X  -146.549, Y  +735.713, Z    +0.000, E1   -53.293, E3 +8210.543}
SPL {X  -144.128, Y  +740.978, Z    +0.000, E1   -52.835, E3 +8220.506}
SPL {X  -141.140, Y  +746.862, Z    +0.000, E1   -52.272, E3 +8231.793}
SPL {X  -128.473, Y  +766.865, Z    +0.000, E1   -45.208, E3 +8326.003}
ENDSPLINE

SPLINE
SPL {X  -149.609, Y  +728.220, Z    +0.000, E1   -30.103, E3 +8411.695}
SPL {X  -157.346, Y  +700.520, Z    +0.000, E1   -17.449, E3 +8426.416}
SPL {X  -159.391, Y  +685.442, Z    +0.000, E1    -8.940, E3 +8430.301}
SPL {X  -159.974, Y  +674.384, Z    +0.000, E1    -1.914, E3 +8431.653}
SPL {X  -160.000, Y  +668.854, Z    +0.000, E1    +3.008, E3 +8432.004}
SPL {X  -160.000, Y  +662.175, Z    +0.000, E1   +11.518, E3 +8432.775}
SPL {X  -160.000, Y  +654.447, Z    +0.000, E1   +21.734, E3 +8434.401}
SPL {X  -160.000, Y  +641.600, Z    +0.000, E1   +35.681, E3 +8438.666}
SPL {X  -160.000, Y  +601.361, Z    +0.000, E1   +52.744, E3 +8462.627}
SPL {X  -160.000, Y  +531.662, Z    +0.000, E1   +56.951, E3 +8534.617}
SPL {X  -160.000, Y  +513.172, Z    +0.000, E1   +56.969, E3 +8560.172}
SPL {X  -160.000, Y  +498.160, Z    +0.000, E1   +56.531, E3 +8583.785}
ENDSPLINE

SPLINE
SPL {X  -160.000, Y  +512.094, Z    +0.000, E1   +49.085, E3 +8607.773}
ENDSPLINE

SPLINE
SPL {X  -160.000, Y  +491.347, Z    +0.000, E1   +50.960, E3 +8633.439}
SPL {X  -160.000, Y  +470.538, Z    +0.000, E1   +52.629, E3 +8658.126}
SPL {X  -160.000, Y  +453.213, Z    +0.000, E1   +53.894, E3 +8677.564}
SPL {X  -160.000, Y  +440.734, Z    +0.000, E1   +54.729, E3 +8691.346}
SPL {X  -160.000, Y  +423.596, Z    +0.000, E1   +55.911, E3 +8709.238}
SPL {X  -160.000, Y  +408.178, Z    +0.000, E1   +56.432, E3 +8727.698}
SPL {X  -160.000, Y  +395.668, Z    +0.000, E1   +56.446, E3 +8745.314}
SPL {X  -159.894, Y  +382.991, Z    +0.000, E1   +56.419, E3 +8763.312}
SPL {X  -159.213, Y  +372.948, Z    +0.000, E1   +56.290, E3 +8778.206}
SPL {X  -158.141, Y  +364.480, Z    +0.000, E1   +56.110, E3 +8791.281}
SPL {X  -156.499, Y  +355.511, Z    +0.000, E1   +55.854, E3 +8805.597}
SPL {X  -154.489, Y  +347.168, Z    +0.000, E1   +55.487, E3 +8819.472}
SPL {X  -152.108, Y  +339.170, Z    +0.000, E1   +55.085, E3 +8833.161}
SPL {X  -149.149, Y  +330.880, Z    +0.000, E1   +54.560, E3 +8847.796}
SPL {X  -146.188, Y  +323.769, Z    +0.000, E1   +53.991, E3 +8860.753}
SPL {X  -143.516, Y  +318.068, Z    +0.000, E1   +53.476, E3 +8871.352}
SPL {X  -140.415, Y  +312.095, Z    +0.000, E1   +52.896, E3 +8882.620}
SPL {X  -128.706, Y  +293.749, Z    +0.000, E1   +44.636, E3 +8984.681}
ENDSPLINE

SPLINE
SPL {X  -149.341, Y  +331.377, Z    +0.000, E1   +30.257, E3 +9064.556}
SPL {X  -155.855, Y  +352.616, Z    +0.000, E1   +20.935, E3 +9076.669}
SPL {X  -158.820, Y  +369.405, Z    +0.000, E1   +11.982, E3 +9082.073}
SPL {X  -159.764, Y  +380.110, Z    +0.000, E1    +5.506, E3 +9083.939}
SPL {X  -159.978, Y  +386.129, Z    +0.000, E1    +1.351, E3 +9084.522}
SPL {X  -160.000, Y  +390.626, Z    +0.000, E1    -2.404, E3 +9084.785}
SPL {X  -160.000, Y  +397.252, Z    +0.000, E1   -10.844, E3 +9085.486}
SPL {X  -160.000, Y  +404.580, Z    +0.000, E1   -20.626, E3 +9086.912}
SPL {X  -160.000, Y  +414.518, Z    +0.000, E1   -32.156, E3 +9090.002}
SPL {X  -160.000, Y  +450.190, Z    +0.000, E1   -50.789, E3 +9110.088}
SPL {X  -160.000, Y  +522.988, Z    +0.000, E1   -55.744, E3 +9188.423}
SPL {X  -160.000, Y  +538.972, Z    +0.000, E1   -55.709, E3 +9211.655}
SPL {X  -160.000, Y  +554.704, Z    +0.000, E1   -55.732, E3 +9234.421}
SPL {X  -160.000, Y  +570.552, Z    +0.000, E1   -55.716, E3 +9257.436}
SPL {X  -160.000, Y  +586.464, Z    +0.000, E1   -55.733, E3 +9280.481}
SPL {X  -160.000, Y  +602.947, Z    +0.000, E1   -55.730, E3 +9304.378}
SPL {X  -160.000, Y  +618.907, Z    +0.000, E1   -55.724, E3 +9327.516}
SPL {X  -160.000, Y  +633.674, Z    +0.000, E1   -55.717, E3 +9348.936}
SPL {X  -160.000, Y  +646.135, Z    +0.000, E1   -55.674, E3 +9367.076}
SPL {X  -160.000, Y  +658.587, Z    +0.000, E1   -55.708, E3 +9385.072}
SPL {X  -160.000, Y  +671.750, Z    +0.000, E1   -55.695, E3 +9404.157}
SPL {X  -159.611, Y  +682.650, Z    +0.000, E1   -55.614, E3 +9420.395}
SPL {X  -158.677, Y  +692.037, Z    +0.000, E1   -55.461, E3 +9434.978}
SPL {X  -157.091, Y  +701.873, Z    +0.000, E1   -55.210, E3 +9450.864}
SPL {X  -154.891, Y  +711.608, Z    +0.000, E1   -54.831, E3 +9467.251}
SPL {X  -152.273, Y  +720.623, Z    +0.000, E1   -54.369, E3 +9482.989}
SPL {X  -149.300, Y  +729.027, Z    +0.000, E1   -53.836, E3 +9498.124}
SPL {X  -146.549, Y  +735.713, Z    +0.000, E1   -53.293, E3 +9510.539}
SPL {X  -144.128, Y  +740.978, Z    +0.000, E1   -52.835, E3 +9520.502}
SPL {X  -141.140, Y  +746.862, Z    +0.000, E1   -52.272, E3 +9531.789}
SPL {X  -128.473, Y  +766.865, Z    +0.000, E1   -45.208, E3 +9625.999}
ENDSPLINE

SPLINE
SPL {X  -149.609, Y  +728.220, Z    +0.000, E1   -30.103, E3 +9711.692}
SPL {X  -157.346, Y  +700.520, Z    +0.000, E1   -17.449, E3 +9726.413}
SPL {X  -159.391, Y  +685.442, Z    +0.000, E1    -8.940, E3 +9730.298}
SPL {X  -159.974, Y  +674.384, Z    +0.000, E1    -1.914, E3 +9731.649}
SPL {X  -160.000, Y  +668.854, Z    +0.000, E1    +3.008, E3 +9732.000}
SPL {X  -160.000, Y  +662.175, Z    +0.000, E1   +11.518, E3 +9732.771}
SPL {X  -160.000, Y  +654.447, Z    +0.000, E1   +21.734, E3 +9734.397}
SPL {X  -160.000, Y  +641.600, Z    +0.000, E1   +35.681, E3 +9738.662}
SPL {X  -160.000, Y  +601.361, Z    +0.000, E1   +52.744, E3 +9762.624}
SPL {X  -160.000, Y  +531.662, Z    +0.000, E1   +56.951, E3 +9834.613}
SPL {X  -160.000, Y  +513.172, Z    +0.000, E1   +56.969, E3 +9860.168}
SPL {X  -160.000, Y  +498.160, Z    +0.000, E1   +56.531, E3 +9883.781}
ENDSPLINE

SPLINE
SPL {X  -160.000, Y  +512.094, Z    +0.000, E1   +49.085, E3 +9907.769}
ENDSPLINE

SPLINE
SPL {X  -160.000, Y  +491.347, Z    +0.000, E1   +50.960, E3 +9933.436}
SPL {X  -160.000, Y  +470.538, Z    +0.000, E1   +52.629, E3 +9958.122}
SPL {X  -160.000, Y  +453.213, Z    +0.000, E1   +53.894, E3 +9977.560}
SPL {X  -160.000, Y  +440.734, Z    +0.000, E1   +54.729, E3 +9991.342}
SPL {X  -160.000, Y  +423.596, Z    +0.000, E1   +55.911, E3 +10009.234}
SPL {X  -160.000, Y  +408.178, Z    +0.000, E1   +56.432, E3 +10027.695}
SPL {X  -160.000, Y  +395.668, Z    +0.000, E1   +56.446, E3 +10045.310}
SPL {X  -159.894, Y  +382.991, Z    +0.000, E1   +56.419, E3 +10063.308}
SPL {X  -159.213, Y  +372.948, Z    +0.000, E1   +56.290, E3 +10078.203}
SPL {X  -158.141, Y  +364.480, Z    +0.000, E1   +56.110, E3 +10091.277}
SPL {X  -156.499, Y  +355.511, Z    +0.000, E1   +55.854, E3 +10105.593}
SPL {X  -154.489, Y  +347.168, Z    +0.000, E1   +55.487, E3 +10119.468}
SPL {X  -152.108, Y  +339.170, Z    +0.000, E1   +55.085, E3 +10133.157}
SPL {X  -149.149, Y  +330.880, Z    +0.000, E1   +54.560, E3 +10147.793}
SPL {X  -146.188, Y  +323.769, Z    +0.000, E1   +53.991, E3 +10160.749}
SPL {X  -143.516, Y  +318.068, Z    +0.000, E1   +53.476, E3 +10171.349}
SPL {X  -140.415, Y  +312.095, Z    +0.000, E1   +52.896, E3 +10182.616}
SPL {X  -128.706, Y  +293.749, Z    +0.000, E1   +44.636, E3 +10284.677}
ENDSPLINE

SPLINE
SPL {X  -149.341, Y  +331.377, Z    +0.000, E1   +30.257, E3 +10364.552}
SPL {X  -155.855, Y  +352.616, Z    +0.000, E1   +20.935, E3 +10376.665}
SPL {X  -158.820, Y  +369.405, Z    +0.000, E1   +11.982, E3 +10382.069}
SPL {X  -159.764, Y  +380.110, Z    +0.000, E1    +5.506, E3 +10383.936}
SPL {X  -159.978, Y  +386.129, Z    +0.000, E1    +1.351, E3 +10384.518}
SPL {X  -160.000, Y  +390.626, Z    +0.000, E1    -2.404, E3 +10384.782}
SPL {X  -160.000, Y  +397.252, Z    +0.000, E1   -10.844, E3 +10385.483}
SPL {X  -160.000, Y  +404.580, Z    +0.000, E1   -20.626, E3 +10386.908}
SPL {X  -160.000, Y  +414.518, Z    +0.000, E1   -32.156, E3 +10389.999}
SPL {X  -160.000, Y  +450.190, Z    +0.000, E1   -50.789, E3 +10410.085}
SPL {X  -160.000, Y  +522.988, Z    +0.000, E1   -55.744, E3 +10488.419}
SPL {X  -160.000, Y  +538.972, Z    +0.000, E1   -55.709, E3 +10511.651}
SPL {X  -160.000, Y  +554.704, Z    +0.000, E1   -55.732, E3 +10534.418}
SPL {X  -160.000, Y  +570.552, Z    +0.000, E1   -55.716, E3 +10557.432}
SPL {X  -160.000, Y  +586.464, Z    +0.000, E1   -55.733, E3 +10580.477}
SPL {X  -160.000, Y  +602.947, Z    +0.000, E1   -55.730, E3 +10604.374}
SPL {X  -160.000, Y  +618.907, Z    +0.000, E1   -55.724, E3 +10627.512}
SPL {X  -160.000, Y  +633.674, Z    +0.000, E1   -55.717, E3 +10648.932}
SPL {X  -160.000, Y  +646.135, Z    +0.000, E1   -55.674, E3 +10667.073}
SPL {X  -160.000, Y  +658.587, Z    +0.000, E1   -55.708, E3 +10685.069}
SPL {X  -160.000, Y  +671.750, Z    +0.000, E1   -55.695, E3 +10704.153}
SPL {X  -159.611, Y  +682.650, Z    +0.000, E1   -55.614, E3 +10720.391}
SPL {X  -158.677, Y  +692.037, Z    +0.000, E1   -55.461, E3 +10734.974}
SPL {X  -157.091, Y  +701.873, Z    +0.000, E1   -55.210, E3 +10750.860}
SPL {X  -154.891, Y  +711.608, Z    +0.000, E1   -54.831, E3 +10767.247}
SPL {X  -152.273, Y  +720.623, Z    +0.000, E1   -54.369, E3 +10782.985}
SPL {X  -149.300, Y  +729.027, Z    +0.000, E1   -53.836, E3 +10798.121}
SPL {X  -146.549, Y  +735.713, Z    +0.000, E1   -53.293, E3 +10810.536}
SPL {X  -144.128, Y  +740.978, Z    +0.000, E1   -52.835, E3 +10820.498}
SPL {X  -141.140, Y  +746.862, Z    +0.000, E1   -52.272, E3 +10831.786}
SPL {X  -128.473, Y  +766.865, Z    +0.000, E1   -45.208, E3 +10925.995}
ENDSPLINE

SPLINE
SPL {X  -149.609, Y  +728.220, Z    +0.000, E1   -30.103, E3 +11011.688}
SPL {X  -157.346, Y  +700.520, Z    +0.000, E1   -17.449, E3 +11026.409}
SPL {X  -159.391, Y  +685.442, Z    +0.000, E1    -8.940, E3 +11030.294}
SPL {X  -159.974, Y  +674.384, Z    +0.000, E1    -1.914, E3 +11031.646}
SPL {X  -160.000, Y  +668.854, Z    +0.000, E1    +3.008, E3 +11031.997}
SPL {X  -160.000, Y  +662.175, Z    +0.000, E1   +11.518, E3 +11032.768}
SPL {X  -160.000, Y  +654.447, Z    +0.000, E1   +21.734, E3 +11034.393}
SPL {X  -160.000, Y  +641.600, Z    +0.000, E1   +35.681, E3 +11038.658}
SPL {X  -160.000, Y  +601.361, Z    +0.000, E1   +52.744, E3 +11062.620}
SPL {X  -160.000, Y  +531.662, Z    +0.000, E1   +56.951, E3 +11134.609}
SPL {X  -160.000, Y  +513.172, Z    +0.000, E1   +56.969, E3 +11160.165}
SPL {X  -160.000, Y  +498.160, Z    +0.000, E1   +56.531, E3 +11183.778}
ENDSPLINE

SPLINE
SPL {X  -160.000, Y  +512.094, Z    +0.000, E1   +49.085, E3 +11207.766}
ENDSPLINE

SPLINE
SPL {X  -160.000, Y  +491.347, Z    +0.000, E1   +50.960, E3 +11233.432}
SPL {X  -160.000, Y  +470.538, Z    +0.000, E1   +52.629, E3 +11258.118}
SPL {X  -160.000, Y  +453.213, Z    +0.000, E1   +53.894, E3 +11277.556}
SPL {X  -160.000, Y  +440.734, Z    +0.000, E1   +54.729, E3 +11291.338}
SPL {X  -160.000, Y  +423.596, Z    +0.000, E1   +55.911, E3 +11309.230}
SPL {X  -160.000, Y  +408.178, Z    +0.000, E1   +56.432, E3 +11327.691}
SPL {X  -160.000, Y  +395.668, Z    +0.000, E1   +56.446, E3 +11345.307}
SPL {X  -159.894, Y  +382.991, Z    +0.000, E1   +56.419, E3 +11363.305}
SPL {X  -159.213, Y  +372.948, Z    +0.000, E1   +56.290, E3 +11378.199}
SPL {X  -158.141, Y  +364.480, Z    +0.000, E1   +56.110, E3 +11391.274}
SPL {X  -156.499, Y  +355.511, Z    +0.000, E1   +55.854, E3 +11405.590}
SPL {X  -154.489, Y  +347.168, Z    +0.000, E1   +55.487, E3 +11419.464}
SPL {X  -152.108, Y  +339.170, Z    +0.000, E1   +55.085, E3 +11433.153}
SPL {X  -149.149, Y  +330.880, Z    +0.000, E1   +54.560, E3 +11447.789}
SPL {X  -146.188, Y  +323.769, Z    +0.000, E1   +53.991, E3 +11460.746}
SPL {X  -143.516, Y  +318.068, Z    +0.000, E1   +53.476, E3 +11471.345}
SPL {X  -140.415, Y  +312.095, Z    +0.000, E1   +52.896, E3 +11482.613}
SPL {X  -128.706, Y  +293.749, Z    +0.000, E1   +44.636, E3 +11584.673}
ENDSPLINE

SPLINE
SPL {X  -149.341, Y  +331.377, Z    +0.000, E1   +30.257, E3 +11664.549}
SPL {X  -155.855, Y  +352.616, Z    +0.000, E1   +20.935, E3 +11676.662}
SPL {X  -158.820, Y  +369.405, Z    +0.000, E1   +11.982, E3 +11682.065}
SPL {X  -159.764, Y  +380.110, Z    +0.000, E1    +5.506, E3 +11683.932}
SPL {X  -159.978, Y  +386.129, Z    +0.000, E1    +1.351, E3 +11684.514}
SPL {X  -160.000, Y  +390.626, Z    +0.000, E1    -2.404, E3 +11684.778}
SPL {X  -160.000, Y  +397.252, Z    +0.000, E1   -10.844, E3 +11685.479}
SPL {X  -160.000, Y  +404.580, Z    +0.000, E1   -20.626, E3 +11686.905}
SPL {X  -160.000, Y  +414.518, Z    +0.000, E1   -32.156, E3 +11689.995}
SPL {X  -160.000, Y  +450.190, Z    +0.000, E1   -50.789, E3 +11710.081}
SPL {X  -160.000, Y  +522.988, Z    +0.000, E1   -55.744, E3 +11788.415}
SPL {X  -160.000, Y  +538.972, Z    +0.000, E1   -55.709, E3 +11811.647}
SPL {X  -160.000, Y  +554.704, Z    +0.000, E1   -55.732, E3 +11834.414}
SPL {X  -160.000, Y  +570.552, Z    +0.000, E1   -55.716, E3 +11857.429}
SPL {X  -160.000, Y  +586.464, Z    +0.000, E1   -55.733, E3 +11880.474}
SPL {X  -160.000, Y  +602.947, Z    +0.000, E1   -55.730, E3 +11904.371}
SPL {X  -160.000, Y  +618.907, Z    +0.000, E1   -55.724, E3 +11927.508}
SPL {X  -160.000, Y  +633.674, Z    +0.000, E1   -55.717, E3 +11948.928}
SPL {X  -160.000, Y  +646.135, Z    +0.000, E1   -55.674, E3 +11967.069}
SPL {X  -160.000, Y  +658.587, Z    +0.000, E1   -55.708, E3 +11985.065}
SPL {X  -160.000, Y  +671.750, Z    +0.000, E1   -55.695, E3 +12004.150}
SPL {X  -159.611, Y  +682.650, Z    +0.000, E1   -55.614, E3 +12020.388}
SPL {X  -158.677, Y  +692.037, Z    +0.000, E1   -55.461, E3 +12034.971}
SPL {X  -157.091, Y  +701.873, Z    +0.000, E1   -55.210, E3 +12050.857}
SPL {X  -154.891, Y  +711.608, Z    +0.000, E1   -54.831, E3 +12067.244}
SPL {X  -152.273, Y  +720.623, Z    +0.000, E1   -54.369, E3 +12082.981}
SPL {X  -149.300, Y  +729.027, Z    +0.000, E1   -53.836, E3 +12098.117}
SPL {X  -146.549, Y  +735.713, Z    +0.000, E1   -53.293, E3 +12110.532}
SPL {X  -144.128, Y  +740.978, Z    +0.000, E1   -52.835, E3 +12120.495}
SPL {X  -141.140, Y  +746.862, Z    +0.000, E1   -52.272, E3 +12131.782}
SPL {X  -128.473, Y  +766.865, Z    +0.000, E1   -45.208, E3 +12225.992}
ENDSPLINE

SPLINE
SPL {X  -149.609, Y  +728.220, Z    +0.000, E1   -30.103, E3 +12311.684}
SPL {X  -157.346, Y  +700.520, Z    +0.000, E1   -17.449, E3 +12326.405}
SPL {X  -159.391, Y  +685.442, Z    +0.000, E1    -8.940, E3 +12330.290}
SPL {X  -159.974, Y  +674.384, Z    +0.000, E1    -1.914, E3 +12331.642}
SPL {X  -160.000, Y  +668.854, Z    +0.000, E1    +3.008, E3 +12331.993}
SPL {X  -160.000, Y  +662.175, Z    +0.000, E1   +11.518, E3 +12332.764}
SPL {X  -160.000, Y  +654.447, Z    +0.000, E1   +21.734, E3 +12334.390}
SPL {X  -160.000, Y  +641.600, Z    +0.000, E1   +35.681, E3 +12338.655}
SPL {X  -160.000, Y  +601.361, Z    +0.000, E1   +52.744, E3 +12362.616}
SPL {X  -160.000, Y  +531.662, Z    +0.000, E1   +56.951, E3 +12434.606}
SPL {X  -160.000, Y  +513.172, Z    +0.000, E1   +56.969, E3 +12460.161}
SPL {X  -160.000, Y  +498.160, Z    +0.000, E1   +56.531, E3 +12483.774}
ENDSPLINE

SPLINE
SPL {X  -160.000, Y  +512.094, Z    +0.000, E1   +49.085, E3 +12507.762}
ENDSPLINE

SPLINE
SPL {X  -160.000, Y  +491.347, Z    +0.000, E1   +50.960, E3 +12533.429}
SPL {X  -160.000, Y  +470.538, Z    +0.000, E1   +52.629, E3 +12558.115}
SPL {X  -160.000, Y  +453.213, Z    +0.000, E1   +53.894, E3 +12577.553}
SPL {X  -160.000, Y  +440.734, Z    +0.000, E1   +54.729, E3 +12591.335}
SPL {X  -160.000, Y  +423.596, Z    +0.000, E1   +55.911, E3 +12609.227}
SPL {X  -160.000, Y  +408.178, Z    +0.000, E1   +56.432, E3 +12627.688}
SPL {X  -160.000, Y  +395.668, Z    +0.000, E1   +56.446, E3 +12645.303}
SPL {X  -159.894, Y  +382.991, Z    +0.000, E1   +56.419, E3 +12663.301}
SPL {X  -159.213, Y  +372.948, Z    +0.000, E1   +56.290, E3 +12678.195}
SPL {X  -158.141, Y  +364.480, Z    +0.000, E1   +56.110, E3 +12691.270}
SPL {X  -156.499, Y  +355.511, Z    +0.000, E1   +55.854, E3 +12705.586}
SPL {X  -154.489, Y  +347.168, Z    +0.000, E1   +55.487, E3 +12719.461}
SPL {X  -152.108, Y  +339.170, Z    +0.000, E1   +55.085, E3 +12733.150}
SPL {X  -149.149, Y  +330.880, Z    +0.000, E1   +54.560, E3 +12747.785}
SPL {X  -146.188, Y  +323.769, Z    +0.000, E1   +53.991, E3 +12760.742}
SPL {X  -143.516, Y  +318.068, Z    +0.000, E1   +53.476, E3 +12771.342}
SPL {X  -140.415, Y  +312.095, Z    +0.000, E1   +52.896, E3 +12782.609}
SPL {X  -128.706, Y  +293.749, Z    +0.000, E1   +44.636, E3 +12884.670}
ENDSPLINE

SPLINE
SPL {X  -149.341, Y  +331.377, Z    +0.000, E1   +30.257, E3 +12964.545}
SPL {X  -155.855, Y  +352.616, Z    +0.000, E1   +20.935, E3 +12976.658}
SPL {X  -158.820, Y  +369.405, Z    +0.000, E1   +11.982, E3 +12982.062}
SPL {X  -159.764, Y  +380.110, Z    +0.000, E1    +5.506, E3 +12983.928}
SPL {X  -159.978, Y  +386.129, Z    +0.000, E1    +1.351, E3 +12984.511}
SPL {X  -160.000, Y  +390.626, Z    +0.000, E1    -2.404, E3 +12984.774}
SPL {X  -160.000, Y  +397.252, Z    +0.000, E1   -10.844, E3 +12985.475}
SPL {X  -160.000, Y  +404.580, Z    +0.000, E1   -20.626, E3 +12986.901}
SPL {X  -160.000, Y  +414.518, Z    +0.000, E1   -32.156, E3 +12989.992}
SPL {X  -160.000, Y  +450.190, Z    +0.000, E1   -50.789, E3 +13010.077}
SPL {X  -160.000, Y  +522.988, Z    +0.000, E1   -55.744, E3 +13088.412}
SPL {X  -160.000, Y  +538.972, Z    +0.000, E1   -55.709, E3 +13111.644}
SPL {X  -160.000, Y  +554.704, Z    +0.000, E1   -55.732, E3 +13134.410}
SPL {X  -160.000, Y  +570.552, Z    +0.000, E1   -55.716, E3 +13157.425}
SPL {X  -160.000, Y  +586.464, Z    +0.000, E1   -55.733, E3 +13180.470}
SPL {X  -160.000, Y  +602.947, Z    +0.000, E1   -55.730, E3 +13204.367}
SPL {X  -160.000, Y  +618.907, Z    +0.000, E1   -55.724, E3 +13227.505}
SPL {X  -160.000, Y  +633.674, Z    +0.000, E1   -55.717, E3 +13248.925}
SPL {X  -160.000, Y  +646.135, Z    +0.000, E1   -55.674, E3 +13267.065}
SPL {X  -160.000, Y  +658.587, Z    +0.000, E1   -55.708, E3 +13285.061}
SPL {X  -160.000, Y  +671.750, Z    +0.000, E1   -55.695, E3 +13304.146}
SPL {X  -159.611, Y  +682.650, Z    +0.000, E1   -55.614, E3 +13320.384}
SPL {X  -158.677, Y  +692.037, Z    +0.000, E1   -55.461, E3 +13334.967}
SPL {X  -157.091, Y  +701.873, Z    +0.000, E1   -55.210, E3 +13350.853}
SPL {X  -154.891, Y  +711.608, Z    +0.000, E1   -54.831, E3 +13367.240}
SPL {X  -152.273, Y  +720.623, Z    +0.000, E1   -54.369, E3 +13382.978}
SPL {X  -149.300, Y  +729.027, Z    +0.000, E1   -53.836, E3 +13398.114}
SPL {X  -146.549, Y  +735.713, Z    +0.000, E1   -53.293, E3 +13410.528}
SPL {X  -144.128, Y  +740.978, Z    +0.000, E1   -52.835, E3 +13420.491}
SPL {X  -141.140, Y  +746.862, Z    +0.000, E1   -52.272, E3 +13431.779}
SPL {X  -128.473, Y  +766.865, Z    +0.000, E1   -45.208, E3 +13525.988}
ENDSPLINE

SPLINE
SPL {X  -149.609, Y  +728.220, Z    +0.000, E1   -30.103, E3 +13611.681}
SPL {X  -157.346, Y  +700.520, Z    +0.000, E1   -17.449, E3 +13626.402}
SPL {X  -159.391, Y  +685.442, Z    +0.000, E1    -8.940, E3 +13630.287}
SPL {X  -159.974, Y  +674.384, Z    +0.000, E1    -1.914, E3 +13631.638}
SPL {X  -160.000, Y  +668.854, Z    +0.000, E1    +3.008, E3 +13631.989}
SPL {X  -160.000, Y  +662.175, Z    +0.000, E1   +11.518, E3 +13632.760}
SPL {X  -160.000, Y  +654.447, Z    +0.000, E1   +21.734, E3 +13634.386}
SPL {X  -160.000, Y  +641.600, Z    +0.000, E1   +35.681, E3 +13638.651}
SPL {X  -160.000, Y  +601.361, Z    +0.000, E1   +52.744, E3 +13662.613}
SPL {X  -160.000, Y  +531.662, Z    +0.000, E1   +56.951, E3 +13734.602}
SPL {X  -160.000, Y  +513.172, Z    +0.000, E1   +56.969, E3 +13760.158}
SPL {X  -160.000, Y  +498.160, Z    +0.000, E1   +56.531, E3 +13783.770}
ENDSPLINE

SPLINE
SPL {X  -160.000, Y  +512.094, Z    +0.000, E1   +49.085, E3 +13807.758}
ENDSPLINE

SPLINE
SPL {X  -160.000, Y  +491.347, Z    +0.000, E1   +50.960, E3 +13833.425}
SPL {X  -160.000, Y  +470.538, Z    +0.000, E1   +52.629, E3 +13858.111}
SPL {X  -160.000, Y  +453.213, Z    +0.000, E1   +53.894, E3 +13877.549}
SPL {X  -160.000, Y  +440.734, Z    +0.000, E1   +54.729, E3 +13891.331}
SPL {X  -160.000, Y  +423.596, Z    +0.000, E1   +55.911, E3 +13909.223}
SPL {X  -160.000, Y  +408.178, Z    +0.000, E1   +56.432, E3 +13927.684}
SPL {X  -160.000, Y  +395.668, Z    +0.000, E1   +56.446, E3 +13945.299}
SPL {X  -159.894, Y  +382.991, Z    +0.000, E1   +56.419, E3 +13963.297}
SPL {X  -159.213, Y  +372.948, Z    +0.000, E1   +56.290, E3 +13978.192}
SPL {X  -158.141, Y  +364.480, Z    +0.000, E1   +56.110, E3 +13991.266}
SPL {X  -156.499, Y  +355.511, Z    +0.000, E1   +55.854, E3 +14005.582}
SPL {X  -154.489, Y  +347.168, Z    +0.000, E1   +55.487, E3 +14019.457}
SPL {X  -152.108, Y  +339.170, Z    +0.000, E1   +55.085, E3 +14033.146}
SPL {X  -149.149, Y  +330.880, Z    +0.000, E1   +54.560, E3 +14047.782}
SPL {X  -146.188, Y  +323.769, Z    +0.000, E1   +53.991, E3 +14060.738}
SPL {X  -143.516, Y  +318.068, Z    +0.000, E1   +53.476, E3 +14071.338}
SPL {X  -140.415, Y  +312.095, Z    +0.000, E1   +52.896, E3 +14082.605}
SPL {X  -128.706, Y  +293.749, Z    +0.000, E1   +44.636, E3 +14184.666}
ENDSPLINE

SPLINE
SPL {X  -149.341, Y  +331.377, Z    +0.000, E1   +30.257, E3 +14264.542}
SPL {X  -155.855, Y  +352.616, Z    +0.000, E1   +20.935, E3 +14276.654}
SPL {X  -158.820, Y  +369.405, Z    +0.000, E1   +11.982, E3 +14282.058}
SPL {X  -159.764, Y  +380.110, Z    +0.000, E1    +5.506, E3 +14283.925}
SPL {X  -159.978, Y  +386.129, Z    +0.000, E1    +1.351, E3 +14284.507}
SPL {X  -160.000, Y  +390.626, Z    +0.000, E1    -2.404, E3 +14284.771}
SPL {X  -160.000, Y  +397.252, Z    +0.000, E1   -10.844, E3 +14285.472}
SPL {X  -160.000, Y  +404.580, Z    +0.000, E1   -20.626, E3 +14286.897}
SPL {X  -160.000, Y  +414.518, Z    +0.000, E1   -32.156, E3 +14289.988}
SPL {X  -160.000, Y  +450.190, Z    +0.000, E1   -50.789, E3 +14310.074}
SPL {X  -160.000, Y  +522.988, Z    +0.000, E1   -55.744, E3 +14388.408}
SPL {X  -160.000, Y  +538.972, Z    +0.000, E1   -55.709, E3 +14411.640}
SPL {X  -160.000, Y  +554.704, Z    +0.000, E1   -55.732, E3 +14434.407}
SPL {X  -160.000, Y  +570.552, Z    +0.000, E1   -55.716, E3 +14457.421}
SPL {X  -160.000, Y  +586.464, Z    +0.000, E1   -55.733, E3 +14480.467}
SPL {X  -160.000, Y  +602.947, Z    +0.000, E1   -55.730, E3 +14504.363}
SPL {X  -160.000, Y  +618.907, Z    +0.000, E1   -55.724, E3 +14527.501}
SPL {X  -160.000, Y  +633.674, Z    +0.000, E1   -55.717, E3 +14548.921}
SPL {X  -160.000, Y  +646.135, Z    +0.000, E1   -55.674, E3 +14567.062}
SPL {X  -160.000, Y  +658.587, Z    +0.000, E1   -55.708, E3 +14585.058}
SPL {X  -160.000, Y  +671.750, Z    +0.000, E1   -55.695, E3 +14604.142}
SPL {X  -159.611, Y  +682.650, Z    +0.000, E1   -55.614, E3 +14620.380}
SPL {X  -158.677, Y  +692.037, Z    +0.000, E1   -55.461, E3 +14634.963}
SPL {X  -157.091, Y  +701.873, Z    +0.000, E1   -55.210, E3 +14650.850}
SPL {X  -154.891, Y  +711.608, Z    +0.000, E1   -54.831, E3 +14667.236}
SPL {X  -152.273, Y  +720.623, Z    +0.000, E1   -54.369, E3 +14682.974}
SPL {X  -149.300, Y  +729.027, Z    +0.000, E1   -53.836, E3 +14698.110}
SPL {X  -146.549, Y  +735.713, Z    +0.000, E1   -53.293, E3 +14710.525}
SPL {X  -144.128, Y  +740.978, Z    +0.000, E1   -52.835, E3 +14720.487}
SPL {X  -141.140, Y  +746.862, Z    +0.000, E1   -52.272, E3 +14731.775}
SPL {X  -128.473, Y  +766.865, Z    +0.000, E1   -45.208, E3 +14825.984}
ENDSPLINE

SPLINE
SPL {X  -149.609, Y  +728.220, Z    +0.000, E1   -30.103, E3 +14911.677}
SPL {X  -157.346, Y  +700.520, Z    +0.000, E1   -17.449, E3 +14926.398}
SPL {X  -159.391, Y  +685.442, Z    +0.000, E1    -8.940, E3 +14930.283}
SPL {X  -159.974, Y  +674.384, Z    +0.000, E1    -1.914, E3 +14931.635}
SPL {X  -160.000, Y  +668.854, Z    +0.000, E1    +3.008, E3 +14931.986}
SPL {X  -160.000, Y  +662.175, Z    +0.000, E1   +11.518, E3 +14932.757}
SPL {X  -160.000, Y  +654.447, Z    +0.000, E1   +21.734, E3 +14934.382}
SPL {X  -160.000, Y  +641.600, Z    +0.000, E1   +35.681, E3 +14938.647}
SPL {X  -160.000, Y  +601.361, Z    +0.000, E1   +52.744, E3 +14962.609}
SPL {X  -160.000, Y  +531.662, Z    +0.000, E1   +56.951, E3 +15034.598}
SPL {X  -160.000, Y  +513.172, Z    +0.000, E1   +56.969, E3 +15060.154}
SPL {X  -160.000, Y  +498.160, Z    +0.000, E1   +56.531, E3 +15083.767}
ENDSPLINE

SPLINE
SPL {X  -160.000, Y  +512.094, Z    +0.000, E1   +49.085, E3 +15107.755}
ENDSPLINE

SPLINE
SPL {X  -160.000, Y  +491.347, Z    +0.000, E1   +50.960, E3 +15133.421}
SPL {X  -160.000, Y  +470.538, Z    +0.000, E1   +52.629, E3 +15158.107}
SPL {X  -160.000, Y  +453.213, Z    +0.000, E1   +53.894, E3 +15177.545}
SPL {X  -160.000, Y  +440.734, Z    +0.000, E1   +54.729, E3 +15191.327}
SPL {X  -160.000, Y  +423.596, Z    +0.000, E1   +55.911, E3 +15209.219}
SPL {X  -160.000, Y  +408.178, Z    +0.000, E1   +56.432, E3 +15227.680}
SPL {X  -160.000, Y  +395.668, Z    +0.000, E1   +56.446, E3 +15245.296}
SPL {X  -159.894, Y  +382.991, Z    +0.000, E1   +56.419, E3 +15263.294}
SPL {X  -159.213, Y  +372.948, Z    +0.000, E1   +56.290, E3 +15278.188}
SPL {X  -158.141, Y  +364.480, Z    +0.000, E1   +56.110, E3 +15291.263}
SPL {X  -156.499, Y  +355.511, Z    +0.000, E1   +55.854, E3 +15305.579}
SPL {X  -154.489, Y  +347.168, Z    +0.000, E1   +55.487, E3 +15319.453}
SPL {X  -152.108, Y  +339.170, Z    +0.000, E1   +55.085, E3 +15333.142}
SPL {X  -149.149, Y  +330.880, Z    +0.000, E1   +54.560, E3 +15347.778}
SPL {X  -146.188, Y  +323.769, Z    +0.000, E1   +53.991, E3 +15360.735}
SPL {X  -143.516, Y  +318.068, Z    +0.000, E1   +53.476, E3 +15371.334}
SPL {X  -140.415, Y  +312.095, Z    +0.000, E1   +52.896, E3 +15382.602}
SPL {X  -128.706, Y  +293.749, Z    +0.000, E1   +44.636, E3 +15484.662}
ENDSPLINE

SPLINE
SPL {X  -149.341, Y  +331.377, Z    +0.000, E1   +30.257, E3 +15564.538}
SPL {X  -155.855, Y  +352.616, Z    +0.000, E1   +20.935, E3 +15576.651}
SPL {X  -158.820, Y  +369.405, Z    +0.000, E1   +11.982, E3 +15582.055}
SPL {X  -159.764, Y  +380.110, Z    +0.000, E1    +5.506, E3 +15583.921}
SPL {X  -159.978, Y  +386.129, Z    +0.000, E1    +1.351, E3 +15584.503}
SPL {X  -160.000, Y  +390.626, Z    +0.000, E1    -2.404, E3 +15584.767}
SPL {X  -160.000, Y  +397.252, Z    +0.000, E1   -10.844, E3 +15585.468}
SPL {X  -160.000, Y  +404.580, Z    +0.000, E1   -20.626, E3 +15586.894}
SPL {X  -160.000, Y  +414.518, Z    +0.000, E1   -32.156, E3 +15589.984}
SPL {X  -160.000, Y  +450.190, Z    +0.000, E1   -50.789, E3 +15610.070}
SPL {X  -160.000, Y  +522.988, Z    +0.000, E1   -55.744, E3 +15688.404}
SPL {X  -160.000, Y  +538.972, Z    +0.000, E1   -55.709, E3 +15711.637}
SPL {X  -160.000, Y  +554.704, Z    +0.000, E1   -55.732, E3 +15734.403}
SPL {X  -160.000, Y  +570.552, Z    +0.000, E1   -55.716, E3 +15757.418}
SPL {X  -160.000, Y  +586.464, Z    +0.000, E1   -55.733, E3 +15780.463}
SPL {X  -160.000, Y  +602.947, Z    +0.000, E1   -55.730, E3 +15804.360}
SPL {X  -160.000, Y  +618.907, Z    +0.000, E1   -55.724, E3 +15827.498}
SPL {X  -160.000, Y  +633.674, Z    +0.000, E1   -55.717, E3 +15848.917}
SPL {X  -160.000, Y  +646.135, Z    +0.000, E1   -55.674, E3 +15867.058}
SPL {X  -160.000, Y  +658.587, Z    +0.000, E1   -55.708, E3 +15885.054}
SPL {X  -160.000, Y  +671.750, Z    +0.000, E1   -55.695, E3 +15904.139}
SPL {X  -159.611, Y  +682.650, Z    +0.000, E1   -55.614, E3 +15920.377}
SPL {X  -158.677, Y  +692.037, Z    +0.000, E1   -55.461, E3 +15934.960}
SPL {X  -157.091, Y  +701.873, Z    +0.000, E1   -55.210, E3 +15950.846}
SPL {X  -154.891, Y  +711.608, Z    +0.000, E1   -54.831, E3 +15967.233}
SPL {X  -152.273, Y  +720.623, Z    +0.000, E1   -54.369, E3 +15982.970}
SPL {X  -149.300, Y  +729.027, Z    +0.000, E1   -53.836, E3 +15998.106}
SPL {X  -146.549, Y  +735.713, Z    +0.000, E1   -53.293, E3 +16010.521}
SPL {X  -144.128, Y  +740.978, Z    +0.000, E1   -52.835, E3 +16020.484}
SPL {X  -141.140, Y  +746.862, Z    +0.000, E1   -52.272, E3 +16031.771}
SPL {X  -128.473, Y  +766.865, Z    +0.000, E1   -45.208, E3 +16125.981}
ENDSPLINE

SPLINE
SPL {X  -149.609, Y  +728.220, Z    +0.000, E1   -30.103, E3 +16211.674}
SPL {X  -157.346, Y  +700.520, Z    +0.000, E1   -17.449, E3 +16226.394}
SPL {X  -159.391, Y  +685.442, Z    +0.000, E1    -8.940, E3 +16230.279}
SPL {X  -159.974, Y  +674.384, Z    +0.000, E1    -1.914, E3 +16231.631}
SPL {X  -160.000, Y  +668.854, Z    +0.000, E1    +3.008, E3 +16231.982}
SPL {X  -160.000, Y  +662.175, Z    +0.000, E1   +11.518, E3 +16232.753}
SPL {X  -160.000, Y  +654.447, Z    +0.000, E1   +21.734, E3 +16234.379}
SPL {X  -160.000, Y  +641.600, Z    +0.000, E1   +35.681, E3 +16238.644}
SPL {X  -160.000, Y  +601.361, Z    +0.000, E1   +52.744, E3 +16262.606}
SPL {X  -160.000, Y  +531.662, Z    +0.000, E1   +56.951, E3 +16334.595}
SPL {X  -160.000, Y  +513.172, Z    +0.000, E1   +56.969, E3 +16360.150}
SPL {X  -160.000, Y  +498.160, Z    +0.000, E1   +56.531, E3 +16383.763}
ENDSPLINE

SPLINE
SPL {X  -160.000, Y  +512.094, Z    +0.000, E1   +49.085, E3 +16407.751}
ENDSPLINE

SPLINE
SPL {X  -160.000, Y  +491.347, Z    +0.000, E1   +50.960, E3 +16433.418}
SPL {X  -160.000, Y  +470.538, Z    +0.000, E1   +52.629, E3 +16458.104}
SPL {X  -160.000, Y  +453.213, Z    +0.000, E1   +53.894, E3 +16477.542}
SPL {X  -160.000, Y  +440.734, Z    +0.000, E1   +54.729, E3 +16491.324}
SPL {X  -160.000, Y  +423.596, Z    +0.000, E1   +55.911, E3 +16509.216}
SPL {X  -160.000, Y  +408.178, Z    +0.000, E1   +56.432, E3 +16527.677}
SPL {X  -160.000, Y  +395.668, Z    +0.000, E1   +56.446, E3 +16545.292}
SPL {X  -159.894, Y  +382.991, Z    +0.000, E1   +56.419, E3 +16563.290}
SPL {X  -159.213, Y  +372.948, Z    +0.000, E1   +56.290, E3 +16578.185}
SPL {X  -158.141, Y  +364.480, Z    +0.000, E1   +56.110, E3 +16591.259}
SPL {X  -156.499, Y  +355.511, Z    +0.000, E1   +55.854, E3 +16605.575}
SPL {X  -154.489, Y  +347.168, Z    +0.000, E1   +55.487, E3 +16619.450}
SPL {X  -152.108, Y  +339.170, Z    +0.000, E1   +55.085, E3 +16633.139}
SPL {X  -149.149, Y  +330.880, Z    +0.000, E1   +54.560, E3 +16647.775}
SPL {X  -146.188, Y  +323.769, Z    +0.000, E1   +53.991, E3 +16660.731}
SPL {X  -143.516, Y  +318.068, Z    +0.000, E1   +53.476, E3 +16671.331}
SPL {X  -140.415, Y  +312.095, Z    +0.000, E1   +52.896, E3 +16682.598}
SPL {X  -128.706, Y  +293.749, Z    +0.000, E1   +44.636, E3 +16784.659}
ENDSPLINE

SPLINE
SPL {X  -149.341, Y  +331.377, Z    +0.000, E1   +30.257, E3 +16864.534}
SPL {X  -155.855, Y  +352.616, Z    +0.000, E1   +20.935, E3 +16876.647}
SPL {X  -158.820, Y  +369.405, Z    +0.000, E1   +11.982, E3 +16882.051}
SPL {X  -159.764, Y  +380.110, Z    +0.000, E1    +5.506, E3 +16883.917}
SPL {X  -159.978, Y  +386.129, Z    +0.000, E1    +1.351, E3 +16884.500}
SPL {X  -160.000, Y  +390.626, Z    +0.000, E1    -2.404, E3 +16884.764}
SPL {X  -160.000, Y  +397.252, Z    +0.000, E1   -10.844, E3 +16885.465}
SPL {X  -160.000, Y  +404.580, Z    +0.000, E1   -20.626, E3 +16886.890}
SPL {X  -160.000, Y  +414.518, Z    +0.000, E1   -32.156, E3 +16889.981}
SPL {X  -160.000, Y  +450.190, Z    +0.000, E1   -50.789, E3 +16910.066}
SPL {X  -160.000, Y  +522.988, Z    +0.000, E1   -55.744, E3 +16988.401}
SPL {X  -160.000, Y  +538.972, Z    +0.000, E1   -55.709, E3 +17011.633}
SPL {X  -160.000, Y  +554.704, Z    +0.000, E1   -55.732, E3 +17034.399}
SPL {X  -160.000, Y  +570.552, Z    +0.000, E1   -55.716, E3 +17057.414}
SPL {X  -160.000, Y  +586.464, Z    +0.000, E1   -55.733, E3 +17080.459}
SPL {X  -160.000, Y  +602.947, Z    +0.000, E1   -55.730, E3 +17104.356}
SPL {X  -160.000, Y  +618.907, Z    +0.000, E1   -55.724, E3 +17127.494}
SPL {X  -160.000, Y  +633.674, Z    +0.000, E1   -55.717, E3 +17148.914}
SPL {X  -160.000, Y  +646.135, Z    +0.000, E1   -55.674, E3 +17167.054}
SPL {X  -160.000, Y  +658.587, Z    +0.000, E1   -55.708, E3 +17185.050}
SPL {X  -160.000, Y  +671.750, Z    +0.000, E1   -55.695, E3 +17204.135}
SPL {X  -159.611, Y  +682.650, Z    +0.000, E1   -55.614, E3 +17220.373}
SPL {X  -158.677, Y  +692.037, Z    +0.000, E1   -55.461, E3 +17234.956}
SPL {X  -157.091, Y  +701.873, Z    +0.000, E1   -55.210, E3 +17250.842}
SPL {X  -154.891, Y  +711.608, Z    +0.000, E1   -54.831, E3 +17267.229}
SPL {X  -152.273, Y  +720.623, Z    +0.000, E1   -54.369, E3 +17282.967}
SPL {X  -149.300, Y  +729.027, Z    +0.000, E1   -53.836, E3 +17298.103}
SPL {X  -146.549, Y  +735.713, Z    +0.000, E1   -53.293, E3 +17310.517}
SPL {X  -144.128, Y  +740.978, Z    +0.000, E1   -52.835, E3 +17320.480}
SPL {X  -141.140, Y  +746.862, Z    +0.000, E1   -52.272, E3 +17331.768}
SPL {X  -128.473, Y  +766.865, Z    +0.000, E1   -45.208, E3 +17425.977}
ENDSPLINE

SPLINE
SPL {X  -149.609, Y  +728.220, Z    +0.000, E1   -30.103, E3 +17511.670}
SPL {X  -157.346, Y  +700.520, Z    +0.000, E1   -17.449, E3 +17526.391}
SPL {X  -159.391, Y  +685.442, Z    +0.000, E1    -8.940, E3 +17530.276}
SPL {X  -159.974, Y  +674.384, Z    +0.000, E1    -1.914, E3 +17531.628}
SPL {X  -160.000, Y  +668.854, Z    +0.000, E1    +3.008, E3 +17531.979}
SPL {X  -160.000, Y  +662.175, Z    +0.000, E1   +11.518, E3 +17532.749}
SPL {X  -160.000, Y  +654.447, Z    +0.000, E1   +21.734, E3 +17534.375}
SPL {X  -160.000, Y  +641.600, Z    +0.000, E1   +35.681, E3 +17538.640}
SPL {X  -160.000, Y  +601.361, Z    +0.000, E1   +52.744, E3 +17562.602}
SPL {X  -160.000, Y  +531.662, Z    +0.000, E1   +56.951, E3 +17634.591}
SPL {X  -160.000, Y  +513.172, Z    +0.000, E1   +56.969, E3 +17660.147}
SPL {X  -160.000, Y  +498.160, Z    +0.000, E1   +56.531, E3 +17683.760}
ENDSPLINE

SPLINE
SPL {X  -160.000, Y  +512.094, Z    +0.000, E1   +49.085, E3 +17707.747}
ENDSPLINE

SPLINE
SPL {X  -160.000, Y  +491.347, Z    +0.000, E1   +50.960, E3 +17733.414}
SPL {X  -160.000, Y  +470.538, Z    +0.000, E1   +52.629, E3 +17758.100}
SPL {X  -160.000, Y  +453.213, Z    +0.000, E1   +53.894, E3 +17777.538}
SPL {X  -160.000, Y  +440.734, Z    +0.000, E1   +54.729, E3 +17791.320}
SPL {X  -160.000, Y  +423.596, Z    +0.000, E1   +55.911, E3 +17809.212}
SPL {X  -160.000, Y  +408.178, Z    +0.000, E1   +56.432, E3 +17827.673}
SPL {X  -160.000, Y  +395.668, Z    +0.000, E1   +56.446, E3 +17845.288}
SPL {X  -159.894, Y  +382.991, Z    +0.000, E1   +56.419, E3 +17863.287}
SPL {X  -159.213, Y  +372.948, Z    +0.000, E1   +56.290, E3 +17878.181}
SPL {X  -158.141, Y  +364.480, Z    +0.000, E1   +56.110, E3 +17891.255}
SPL {X  -156.499, Y  +355.511, Z    +0.000, E1   +55.854, E3 +17905.572}
SPL {X  -154.489, Y  +347.168, Z    +0.000, E1   +55.487, E3 +17919.446}
SPL {X  -152.108, Y  +339.170, Z    +0.000, E1   +55.085, E3 +17933.135}
SPL {X  -149.149, Y  +330.880, Z    +0.000, E1   +54.560, E3 +17947.771}
SPL {X  -146.188, Y  +323.769, Z    +0.000, E1   +53.991, E3 +17960.728}
SPL {X  -143.516, Y  +318.068, Z    +0.000, E1   +53.476, E3 +17971.327}
SPL {X  -140.415, Y  +312.095, Z    +0.000, E1   +52.896, E3 +17982.595}
SPL {X  -128.706, Y  +293.749, Z    +0.000, E1   +44.636, E3 +18084.655}
ENDSPLINE

SPLINE
SPL {X  -149.341, Y  +331.377, Z    +0.000, E1   +30.257, E3 +18164.531}
SPL {X  -155.855, Y  +352.616, Z    +0.000, E1   +20.935, E3 +18176.644}
SPL {X  -158.820, Y  +369.405, Z    +0.000, E1   +11.982, E3 +18182.047}
SPL {X  -159.764, Y  +380.110, Z    +0.000, E1    +5.506, E3 +18183.914}
SPL {X  -159.978, Y  +386.129, Z    +0.000, E1    +1.351, E3 +18184.496}
SPL {X  -160.000, Y  +390.626, Z    +0.000, E1    -2.404, E3 +18184.760}
SPL {X  -160.000, Y  +397.252, Z    +0.000, E1   -10.844, E3 +18185.461}
SPL {X  -160.000, Y  +404.580, Z    +0.000, E1   -20.626, E3 +18186.887}
SPL {X  -160.000, Y  +414.518, Z    +0.000, E1   -32.156, E3 +18189.977}
SPL {X  -160.000, Y  +450.190, Z    +0.000, E1   -50.789, E3 +18210.063}
SPL {X  -160.000, Y  +522.988, Z    +0.000, E1   -55.744, E3 +18288.397}
SPL {X  -160.000, Y  +538.972, Z    +0.000, E1   -55.709, E3 +18311.629}
SPL {X  -160.000, Y  +554.704, Z    +0.000, E1   -55.732, E3 +18334.396}
SPL {X  -160.000, Y  +570.552, Z    +0.000, E1   -55.716, E3 +18357.411}
SPL {X  -160.000, Y  +586.464, Z    +0.000, E1   -55.733, E3 +18380.456}
SPL {X  -160.000, Y  +602.947, Z    +0.000, E1   -55.730, E3 +18404.352}
SPL {X  -160.000, Y  +618.907, Z    +0.000, E1   -55.724, E3 +18427.490}
SPL {X  -160.000, Y  +633.674, Z    +0.000, E1   -55.717, E3 +18448.910}
SPL {X  -160.000, Y  +646.135, Z    +0.000, E1   -55.674, E3 +18467.051}
SPL {X  -160.000, Y  +658.587, Z    +0.000, E1   -55.708, E3 +18485.047}
SPL {X  -160.000, Y  +671.750, Z    +0.000, E1   -55.695, E3 +18504.132}
SPL {X  -159.611, Y  +682.650, Z    +0.000, E1   -55.614, E3 +18520.370}
SPL {X  -158.677, Y  +692.037, Z    +0.000, E1   -55.461, E3 +18534.952}
SPL {X  -157.091, Y  +701.873, Z    +0.000, E1   -55.210, E3 +18550.839}
SPL {X  -154.891, Y  +711.608, Z    +0.000, E1   -54.831, E3 +18567.226}
SPL {X  -152.273, Y  +720.623, Z    +0.000, E1   -54.369, E3 +18582.963}
SPL {X  -149.300, Y  +729.027, Z    +0.000, E1   -53.836, E3 +18598.099}
SPL {X  -146.549, Y  +735.713, Z    +0.000, E1   -53.293, E3 +18610.514}
SPL {X  -144.128, Y  +740.978, Z    +0.000, E1   -52.835, E3 +18620.477}
SPL {X  -141.140, Y  +746.862, Z    +0.000, E1   -52.272, E3 +18631.764}
SPL {X  -128.473, Y  +766.865, Z    +0.000, E1   -45.208, E3 +18725.974}
ENDSPLINE

SPLINE
SPL {X  -149.609, Y  +728.220, Z    +0.000, E1   -30.103, E3 +18811.666}
SPL {X  -157.346, Y  +700.520, Z    +0.000, E1   -17.449, E3 +18826.387}
SPL {X  -159.391, Y  +685.442, Z    +0.000, E1    -8.940, E3 +18830.272}
SPL {X  -159.974, Y  +674.384, Z    +0.000, E1    -1.914, E3 +18831.624}
SPL {X  -160.000, Y  +668.854, Z    +0.000, E1    +3.008, E3 +18831.975}
SPL {X  -160.000, Y  +662.175, Z    +0.000, E1   +11.518, E3 +18832.746}
SPL {X  -160.000, Y  +654.447, Z    +0.000, E1   +21.734, E3 +18834.371}
SPL {X  -160.000, Y  +641.600, Z    +0.000, E1   +35.681, E3 +18838.636}
SPL {X  -160.000, Y  +601.361, Z    +0.000, E1   +52.744, E3 +18862.598}
SPL {X  -160.000, Y  +531.662, Z    +0.000, E1   +56.951, E3 +18934.588}
SPL {X  -160.000, Y  +513.172, Z    +0.000, E1   +56.969, E3 +18960.143}
SPL {X  -160.000, Y  +498.160, Z    +0.000, E1   +56.531, E3 +18983.756}
ENDSPLINE

SPLINE
SPL {X  -160.000, Y  +512.094, Z    +0.000, E1   +49.085, E3 +19007.744}
ENDSPLINE

SPLINE
SPL {X  -160.000, Y  +491.347, Z    +0.000, E1   +50.960, E3 +19033.410}
SPL {X  -160.000, Y  +470.538, Z    +0.000, E1   +52.629, E3 +19058.097}
SPL {X  -160.000, Y  +453.213, Z    +0.000, E1   +53.894, E3 +19077.535}
SPL {X  -160.000, Y  +440.734, Z    +0.000, E1   +54.729, E3 +19091.317}
SPL {X  -160.000, Y  +423.596, Z    +0.000, E1   +55.911, E3 +19109.209}
SPL {X  -160.000, Y  +408.178, Z    +0.000, E1   +56.432, E3 +19127.669}
SPL {X  -160.000, Y  +395.668, Z    +0.000, E1   +56.446, E3 +19145.285}
SPL {X  -159.894, Y  +382.991, Z    +0.000, E1   +56.419, E3 +19163.283}
SPL {X  -159.213, Y  +372.948, Z    +0.000, E1   +56.290, E3 +19178.177}
SPL {X  -158.141, Y  +364.480, Z    +0.000, E1   +56.110, E3 +19191.252}
SPL {X  -156.499, Y  +355.511, Z    +0.000, E1   +55.854, E3 +19205.568}
SPL {X  -154.489, Y  +347.168, Z    +0.000, E1   +55.487, E3 +19219.442}
SPL {X  -152.108, Y  +339.170, Z    +0.000, E1   +55.085, E3 +19233.132}
SPL {X  -149.149, Y  +330.880, Z    +0.000, E1   +54.560, E3 +19247.767}
SPL {X  -146.188, Y  +323.769, Z    +0.000, E1   +53.991, E3 +19260.724}
SPL {X  -143.516, Y  +318.068, Z    +0.000, E1   +53.476, E3 +19271.323}
SPL {X  -140.415, Y  +312.095, Z    +0.000, E1   +52.896, E3 +19282.591}
SPL {X  -128.706, Y  +293.749, Z    +0.000, E1   +44.636, E3 +19384.652}
ENDSPLINE

SPLINE
SPL {X  -149.341, Y  +331.377, Z    +0.000, E1   +30.257, E3 +19464.527}
SPL {X  -155.855, Y  +352.616, Z    +0.000, E1   +20.935, E3 +19476.640}
SPL {X  -158.820, Y  +369.405, Z    +0.000, E1   +11.982, E3 +19482.044}
SPL {X  -159.764, Y  +380.110, Z    +0.000, E1    +5.506, E3 +19483.910}
SPL {X  -159.978, Y  +386.129, Z    +0.000, E1    +1.351, E3 +19484.493}
SPL {X  -160.000, Y  +390.626, Z    +0.000, E1    -2.404, E3 +19484.756}
SPL {X  -160.000, Y  +397.252, Z    +0.000, E1   -10.844, E3 +19485.457}
SPL {X  -160.000, Y  +404.580, Z    +0.000, E1   -20.626, E3 +19486.883}
SPL {X  -160.000, Y  +414.518, Z    +0.000, E1   -32.156, E3 +19489.973}
SPL {X  -160.000, Y  +450.190, Z    +0.000, E1   -50.789, E3 +19510.059}
SPL {X  -160.000, Y  +522.988, Z    +0.000, E1   -55.744, E3 +19588.394}
SPL {X  -160.000, Y  +538.972, Z    +0.000, E1   -55.709, E3 +19611.626}
SPL {X  -160.000, Y  +554.704, Z    +0.000, E1   -55.732, E3 +19634.392}
SPL {X  -160.000, Y  +570.552, Z    +0.000, E1   -55.716, E3 +19657.407}
SPL {X  -160.000, Y  +586.464, Z    +0.000, E1   -55.733, E3 +19680.452}
SPL {X  -160.000, Y  +602.947, Z    +0.000, E1   -55.730, E3 +19704.349}
SPL {X  -160.000, Y  +618.907, Z    +0.000, E1   -55.724, E3 +19727.487}
SPL {X  -160.000, Y  +633.674, Z    +0.000, E1   -55.717, E3 +19748.907}
SPL {X  -160.000, Y  +646.135, Z    +0.000, E1   -55.674, E3 +19767.047}
SPL {X  -160.000, Y  +658.587, Z    +0.000, E1   -55.708, E3 +19785.043}
SPL {X  -160.000, Y  +671.750, Z    +0.000, E1   -55.695, E3 +19804.128}
SPL {X  -159.611, Y  +682.650, Z    +0.000, E1   -55.614, E3 +19820.366}
SPL {X  -158.677, Y  +692.037, Z    +0.000, E1   -55.461, E3 +19834.949}
SPL {X  -157.091, Y  +701.873, Z    +0.000, E1   -55.210, E3 +19850.835}
SPL {X  -154.891, Y  +711.608, Z    +0.000, E1   -54.831, E3 +19867.222}
SPL {X  -152.273, Y  +720.623, Z    +0.000, E1   -54.369, E3 +19882.959}
SPL {X  -149.300, Y  +729.027, Z    +0.000, E1   -53.836, E3 +19898.095}
SPL {X  -146.549, Y  +735.713, Z    +0.000, E1   -53.293, E3 +19910.510}
SPL {X  -144.128, Y  +740.978, Z    +0.000, E1   -52.835, E3 +19920.473}
SPL {X  -141.140, Y  +746.862, Z    +0.000, E1   -52.272, E3 +19931.760}
SPL {X  -128.473, Y  +766.865, Z    +0.000, E1   -45.208, E3 +20025.970}
ENDSPLINE

SPLINE
SPL {X  -149.609, Y  +728.220, Z    +0.000, E1   -30.103, E3 +20111.663}
SPL {X  -157.346, Y  +700.520, Z    +0.000, E1   -17.449, E3 +20126.384}
SPL {X  -159.391, Y  +685.442, Z    +0.000, E1    -8.940, E3 +20130.269}
SPL {X  -159.974, Y  +674.384, Z    +0.000, E1    -1.914, E3 +20131.620}
SPL {X  -160.000, Y  +668.854, Z    +0.000, E1    +3.008, E3 +20131.971}
SPL {X  -160.000, Y  +662.175, Z    +0.000, E1   +11.518, E3 +20132.742}
SPL {X  -160.000, Y  +654.447, Z    +0.000, E1   +21.734, E3 +20134.368}
SPL {X  -160.000, Y  +641.600, Z    +0.000, E1   +35.681, E3 +20138.633}
SPL {X  -160.000, Y  +601.361, Z    +0.000, E1   +52.744, E3 +20162.595}
SPL {X  -160.000, Y  +531.662, Z    +0.000, E1   +56.951, E3 +20234.584}
SPL {X  -160.000, Y  +513.172, Z    +0.000, E1   +56.969, E3 +20260.139}
SPL {X  -160.000, Y  +498.160, Z    +0.000, E1   +56.531, E3 +20283.752}
ENDSPLINE

SPLINE
SPL {X  -160.000, Y  +512.094, Z    +0.000, E1   +49.085, E3 +20307.740}
ENDSPLINE

SPLINE
SPL {X  -160.000, Y  +491.347, Z    +0.000, E1   +50.960, E3 +20333.407}
SPL {X  -160.000, Y  +470.538, Z    +0.000, E1   +52.629, E3 +20358.093}
SPL {X  -160.000, Y  +453.213, Z    +0.000, E1   +53.894, E3 +20377.531}
SPL {X  -160.000, Y  +440.734, Z    +0.000, E1   +54.729, E3 +20391.313}
SPL {X  -160.000, Y  +423.596, Z    +0.000, E1   +55.911, E3 +20409.205}
SPL {X  -160.000, Y  +408.178, Z    +0.000, E1   +56.432, E3 +20427.666}
SPL {X  -160.000, Y  +395.668, Z    +0.000, E1   +56.446, E3 +20445.281}
SPL {X  -159.894, Y  +382.991, Z    +0.000, E1   +56.419, E3 +20463.279}
SPL {X  -159.213, Y  +372.948, Z    +0.000, E1   +56.290, E3 +20478.174}
SPL {X  -158.141, Y  +364.480, Z    +0.000, E1   +56.110, E3 +20491.248}
SPL {X  -156.499, Y  +355.511, Z    +0.000, E1   +55.854, E3 +20505.564}
SPL {X  -154.489, Y  +347.168, Z    +0.000, E1   +55.487, E3 +20519.439}
SPL {X  -152.108, Y  +339.170, Z    +0.000, E1   +55.085, E3 +20533.128}
SPL {X  -149.149, Y  +330.880, Z    +0.000, E1   +54.560, E3 +20547.764}
SPL {X  -146.188, Y  +323.769, Z    +0.000, E1   +53.991, E3 +20560.720}
SPL {X  -143.516, Y  +318.068, Z    +0.000, E1   +53.476, E3 +20571.320}
SPL {X  -140.415, Y  +312.095, Z    +0.000, E1   +52.896, E3 +20582.587}
SPL {X  -128.706, Y  +293.749, Z    +0.000, E1   +44.636, E3 +20684.648}
ENDSPLINE

SPLINE
SPL {X  -149.341, Y  +331.377, Z    +0.000, E1   +30.257, E3 +20764.523}
SPL {X  -155.855, Y  +352.616, Z    +0.000, E1   +20.935, E3 +20776.636}
SPL {X  -158.820, Y  +369.405, Z    +0.000, E1   +11.982, E3 +20782.040}
SPL {X  -159.764, Y  +380.110, Z    +0.000, E1    +5.506, E3 +20783.906}
SPL {X  -159.978, Y  +386.129, Z    +0.000, E1    +1.351, E3 +20784.489}
SPL {X  -160.000, Y  +390.626, Z    +0.000, E1    -2.404, E3 +20784.753}
SPL {X  -160.000, Y  +397.252, Z    +0.000, E1   -10.844, E3 +20785.454}
SPL {X  -160.000, Y  +404.580, Z    +0.000, E1   -20.626, E3 +20786.879}
SPL {X  -160.000, Y  +414.518, Z    +0.000, E1   -32.156, E3 +20789.970}
SPL {X  -160.000, Y  +450.190, Z    +0.000, E1   -50.789, E3 +20810.056}
SPL {X  -160.000, Y  +522.988, Z    +0.000, E1   -55.744, E3 +20888.390}
SPL {X  -160.000, Y  +538.972, Z    +0.000, E1   -55.709, E3 +20911.622}
SPL {X  -160.000, Y  +554.704, Z    +0.000, E1   -55.732, E3 +20934.389}
SPL {X  -160.000, Y  +570.552, Z    +0.000, E1   -55.716, E3 +20957.403}
SPL {X  -160.000, Y  +586.464, Z    +0.000, E1   -55.733, E3 +20980.448}
SPL {X  -160.000, Y  +602.947, Z    +0.000, E1   -55.730, E3 +21004.345}
SPL {X  -160.000, Y  +618.907, Z    +0.000, E1   -55.724, E3 +21027.483}
SPL {X  -160.000, Y  +633.674, Z    +0.000, E1   -55.717, E3 +21048.903}
SPL {X  -160.000, Y  +646.135, Z    +0.000, E1   -55.674, E3 +21067.044}
SPL {X  -160.000, Y  +658.587, Z    +0.000, E1   -55.708, E3 +21085.040}
SPL {X  -160.000, Y  +671.750, Z    +0.000, E1   -55.695, E3 +21104.124}
SPL {X  -159.611, Y  +682.650, Z    +0.000, E1   -55.614, E3 +21120.362}
SPL {X  -158.677, Y  +692.037, Z    +0.000, E1   -55.461, E3 +21134.945}
SPL {X  -157.091, Y  +701.873, Z    +0.000, E1   -55.210, E3 +21150.831}
SPL {X  -154.891, Y  +711.608, Z    +0.000, E1   -54.831, E3 +21167.218}
SPL {X  -152.273, Y  +720.623, Z    +0.000, E1   -54.369, E3 +21182.956}
SPL {X  -149.300, Y  +729.027, Z    +0.000, E1   -53.836, E3 +21198.092}
SPL {X  -146.549, Y  +735.713, Z    +0.000, E1   -53.293, E3 +21210.507}
SPL {X  -144.128, Y  +740.978, Z    +0.000, E1   -52.835, E3 +21220.469}
SPL {X  -141.140, Y  +746.862, Z    +0.000, E1   -52.272, E3 +21231.757}
SPL {X  -128.473, Y  +766.865, Z    +0.000, E1   -45.208, E3 +21325.966}
ENDSPLINE

SPLINE
SPL {X  -149.609, Y  +728.220, Z    +0.000, E1   -30.103, E3 +21411.659}
SPL {X  -157.346, Y  +700.520, Z    +0.000, E1   -17.449, E3 +21426.380}
SPL {X  -159.391, Y  +685.442, Z    +0.000, E1    -8.940, E3 +21430.265}
SPL {X  -159.974, Y  +674.384, Z    +0.000, E1    -1.914, E3 +21431.617}
SPL {X  -160.000, Y  +668.854, Z    +0.000, E1    +3.008, E3 +21431.968}
SPL {X  -160.000, Y  +662.175, Z    +0.000, E1   +11.518, E3 +21432.738}
SPL {X  -160.000, Y  +654.447, Z    +0.000, E1   +21.734, E3 +21434.364}
SPL {X  -160.000, Y  +641.600, Z    +0.000, E1   +35.681, E3 +21438.629}
SPL {X  -160.000, Y  +601.361, Z    +0.000, E1   +52.744, E3 +21462.591}
SPL {X  -160.000, Y  +531.662, Z    +0.000, E1   +56.951, E3 +21534.580}
SPL {X  -160.000, Y  +513.172, Z    +0.000, E1   +56.969, E3 +21560.136}
SPL {X  -160.000, Y  +498.160, Z    +0.000, E1   +56.531, E3 +21583.749}
ENDSPLINE

SPLINE
SPL {X  -160.000, Y  +512.094, Z    +0.000, E1   +49.085, E3 +21607.737}
ENDSPLINE

SPLINE
SPL {X  -160.000, Y  +491.347, Z    +0.000, E1   +50.960, E3 +21633.403}
SPL {X  -160.000, Y  +470.538, Z    +0.000, E1   +52.629, E3 +21658.089}
SPL {X  -160.000, Y  +453.213, Z    +0.000, E1   +53.894, E3 +21677.527}
SPL {X  -160.000, Y  +440.734, Z    +0.000, E1   +54.729, E3 +21691.309}
SPL {X  -160.000, Y  +423.596, Z    +0.000, E1   +55.911, E3 +21709.201}
SPL {X  -160.000, Y  +408.178, Z    +0.000, E1   +56.432, E3 +21727.662}
SPL {X  -160.000, Y  +395.668, Z    +0.000, E1   +56.446, E3 +21745.277}
SPL {X  -159.894, Y  +382.991, Z    +0.000, E1   +56.419, E3 +21763.276}
SPL {X  -159.213, Y  +372.948, Z    +0.000, E1   +56.290, E3 +21778.170}
SPL {X  -158.141, Y  +364.480, Z    +0.000, E1   +56.110, E3 +21791.245}
SPL {X  -156.499, Y  +355.511, Z    +0.000, E1   +55.854, E3 +21805.561}
SPL {X  -154.489, Y  +347.168, Z    +0.000, E1   +55.487, E3 +21819.435}
SPL {X  -152.108, Y  +339.170, Z    +0.000, E1   +55.085, E3 +21833.124}
SPL {X  -149.149, Y  +330.880, Z    +0.000, E1   +54.560, E3 +21847.760}
SPL {X  -146.188, Y  +323.769, Z    +0.000, E1   +53.991, E3 +21860.717}
SPL {X  -143.516, Y  +318.068, Z    +0.000, E1   +53.476, E3 +21871.316}
SPL {X  -140.415, Y  +312.095, Z    +0.000, E1   +52.896, E3 +21882.584}
SPL {X  -128.706, Y  +293.749, Z    +0.000, E1   +44.636, E3 +21984.644}
ENDSPLINE

SPLINE
SPL {X  -149.341, Y  +331.377, Z    +0.000, E1   +30.257, E3 +22064.520}
SPL {X  -155.855, Y  +352.616, Z    +0.000, E1   +20.935, E3 +22076.633}
SPL {X  -158.820, Y  +369.405, Z    +0.000, E1   +11.982, E3 +22082.036}
SPL {X  -159.764, Y  +380.110, Z    +0.000, E1    +5.506, E3 +22083.903}
SPL {X  -159.978, Y  +386.129, Z    +0.000, E1    +1.351, E3 +22084.485}
SPL {X  -160.000, Y  +390.626, Z    +0.000, E1    -2.404, E3 +22084.749}
SPL {X  -160.000, Y  +397.252, Z    +0.000, E1   -10.844, E3 +22085.450}
SPL {X  -160.000, Y  +404.580, Z    +0.000, E1   -20.626, E3 +22086.876}
SPL {X  -160.000, Y  +414.518, Z    +0.000, E1   -32.156, E3 +22089.966}
SPL {X  -160.000, Y  +450.190, Z    +0.000, E1   -50.789, E3 +22110.052}
SPL {X  -160.000, Y  +522.988, Z    +0.000, E1   -55.744, E3 +22188.386}
SPL {X  -160.000, Y  +538.972, Z    +0.000, E1   -55.709, E3 +22211.618}
SPL {X  -160.000, Y  +554.704, Z    +0.000, E1   -55.732, E3 +22234.385}
SPL {X  -160.000, Y  +570.552, Z    +0.000, E1   -55.716, E3 +22257.400}
SPL {X  -160.000, Y  +586.464, Z    +0.000, E1   -55.733, E3 +22280.445}
SPL {X  -160.000, Y  +602.947, Z    +0.000, E1   -55.730, E3 +22304.342}
SPL {X  -160.000, Y  +618.907, Z    +0.000, E1   -55.724, E3 +22327.479}
SPL {X  -160.000, Y  +633.674, Z    +0.000, E1   -55.717, E3 +22348.899}
SPL {X  -160.000, Y  +646.135, Z    +0.000, E1   -55.674, E3 +22367.040}
SPL {X  -160.000, Y  +658.587, Z    +0.000, E1   -55.708, E3 +22385.036}
SPL {X  -160.000, Y  +671.750, Z    +0.000, E1   -55.695, E3 +22404.121}
SPL {X  -159.611, Y  +682.650, Z    +0.000, E1   -55.614, E3 +22420.359}
SPL {X  -158.677, Y  +692.037, Z    +0.000, E1   -55.461, E3 +22434.942}
SPL {X  -157.091, Y  +701.873, Z    +0.000, E1   -55.210, E3 +22450.828}
SPL {X  -154.891, Y  +711.608, Z    +0.000, E1   -54.831, E3 +22467.215}
SPL {X  -152.273, Y  +720.623, Z    +0.000, E1   -54.369, E3 +22482.952}
SPL {X  -149.300, Y  +729.027, Z    +0.000, E1   -53.836, E3 +22498.088}
SPL {X  -146.549, Y  +735.713, Z    +0.000, E1   -53.293, E3 +22510.503}
SPL {X  -144.128, Y  +740.978, Z    +0.000, E1   -52.835, E3 +22520.466}
SPL {X  -141.140, Y  +746.862, Z    +0.000, E1   -52.272, E3 +22531.753}
SPL {X  -128.473, Y  +766.865, Z    +0.000, E1   -45.208, E3 +22625.963}
ENDSPLINE

SPLINE
SPL {X  -149.609, Y  +728.220, Z    +0.000, E1   -30.103, E3 +22711.655}
SPL {X  -157.346, Y  +700.520, Z    +0.000, E1   -17.449, E3 +22726.376}
SPL {X  -159.391, Y  +685.442, Z    +0.000, E1    -8.940, E3 +22730.261}
SPL {X  -159.974, Y  +674.384, Z    +0.000, E1    -1.914, E3 +22731.613}
SPL {X  -160.000, Y  +668.854, Z    +0.000, E1    +3.008, E3 +22731.964}
SPL {X  -160.000, Y  +662.175, Z    +0.000, E1   +11.518, E3 +22732.735}
SPL {X  -160.000, Y  +654.447, Z    +0.000, E1   +21.734, E3 +22734.361}
SPL {X  -160.000, Y  +641.600, Z    +0.000, E1   +35.681, E3 +22738.626}
SPL {X  -160.000, Y  +601.361, Z    +0.000, E1   +52.744, E3 +22762.587}
SPL {X  -160.000, Y  +531.662, Z    +0.000, E1   +56.951, E3 +22834.577}
SPL {X  -160.000, Y  +513.172, Z    +0.000, E1   +56.969, E3 +22860.132}
SPL {X  -160.000, Y  +498.160, Z    +0.000, E1   +56.531, E3 +22883.745}
ENDSPLINE

SPLINE
SPL {X  -160.000, Y  +512.094, Z    +0.000, E1   +49.085, E3 +22907.733}
ENDSPLINE

SPLINE
SPL {X  -160.000, Y  +491.347, Z    +0.000, E1   +50.960, E3 +22933.400}
SPL {X  -160.000, Y  +470.538, Z    +0.000, E1   +52.629, E3 +22958.086}
SPL {X  -160.000, Y  +453.213, Z    +0.000, E1   +53.894, E3 +22977.524}
SPL {X  -160.000, Y  +440.734, Z    +0.000, E1   +54.729, E3 +22991.306}
SPL {X  -160.000, Y  +423.596, Z    +0.000, E1   +55.911, E3 +23009.198}
SPL {X  -160.000, Y  +408.178, Z    +0.000, E1   +56.432, E3 +23027.659}
SPL {X  -160.000, Y  +395.668, Z    +0.000, E1   +56.446, E3 +23045.274}
SPL {X  -159.894, Y  +382.991, Z    +0.000, E1   +56.419, E3 +23063.272}
SPL {X  -159.213, Y  +372.948, Z    +0.000, E1   +56.290, E3 +23078.166}
SPL {X  -158.141, Y  +364.480, Z    +0.000, E1   +56.110, E3 +23091.241}
SPL {X  -156.499, Y  +355.511, Z    +0.000, E1   +55.854, E3 +23105.557}
SPL {X  -154.489, Y  +347.168, Z    +0.000, E1   +55.487, E3 +23119.432}
SPL {X  -152.108, Y  +339.170, Z    +0.000, E1   +55.085, E3 +23133.121}
SPL {X  -149.149, Y  +330.880, Z    +0.000, E1   +54.560, E3 +23147.756}
SPL {X  -146.188, Y  +323.769, Z    +0.000, E1   +53.991, E3 +23160.713}
SPL {X  -143.516, Y  +318.068, Z    +0.000, E1   +53.476, E3 +23171.313}
SPL {X  -140.415, Y  +312.095, Z    +0.000, E1   +52.896, E3 +23182.580}
SPL {X  -128.706, Y  +293.749, Z    +0.000, E1   +44.636, E3 +23284.641}
ENDSPLINE

SPLINE
SPL {X  -149.341, Y  +331.377, Z    +0.000, E1   +30.257, E3 +23364.516}
SPL {X  -155.855, Y  +352.616, Z    +0.000, E1   +20.935, E3 +23376.629}
SPL {X  -158.820, Y  +369.405, Z    +0.000, E1   +11.982, E3 +23382.033}
SPL {X  -159.764, Y  +380.110, Z    +0.000, E1    +5.506, E3 +23383.899}
SPL {X  -159.978, Y  +386.129, Z    +0.000, E1    +1.351, E3 +23384.482}
SPL {X  -160.000, Y  +390.626, Z    +0.000, E1    -2.404, E3 +23384.745}
SPL {X  -160.000, Y  +397.252, Z    +0.000, E1   -10.844, E3 +23385.446}
SPL {X  -160.000, Y  +404.580, Z    +0.000, E1   -20.626, E3 +23386.872}
SPL {X  -160.000, Y  +414.518, Z    +0.000, E1   -32.156, E3 +23389.963}
SPL {X  -160.000, Y  +450.190, Z    +0.000, E1   -50.789, E3 +23410.048}
SPL {X  -160.000, Y  +522.988, Z    +0.000, E1   -55.744, E3 +23488.383}
SPL {X  -160.000, Y  +538.972, Z    +0.000, E1   -55.709, E3 +23511.615}
SPL {X  -160.000, Y  +554.704, Z    +0.000, E1   -55.732, E3 +23534.381}
SPL {X  -160.000, Y  +570.552, Z    +0.000, E1   -55.716, E3 +23557.396}
SPL {X  -160.000, Y  +586.464, Z    +0.000, E1   -55.733, E3 +23580.441}
SPL {X  -160.000, Y  +602.947, Z    +0.000, E1   -55.730, E3 +23604.338}
SPL {X  -160.000, Y  +618.907, Z    +0.000, E1   -55.724, E3 +23627.476}
SPL {X  -160.000, Y  +633.674, Z    +0.000, E1   -55.717, E3 +23648.896}
SPL {X  -160.000, Y  +646.135, Z    +0.000, E1   -55.674, E3 +23667.036}
SPL {X  -160.000, Y  +658.587, Z    +0.000, E1   -55.708, E3 +23685.032}
SPL {X  -160.000, Y  +671.750, Z    +0.000, E1   -55.695, E3 +23704.117}
SPL {X  -159.611, Y  +682.650, Z    +0.000, E1   -55.614, E3 +23720.355}
SPL {X  -158.677, Y  +692.037, Z    +0.000, E1   -55.461, E3 +23734.938}
SPL {X  -157.091, Y  +701.873, Z    +0.000, E1   -55.210, E3 +23750.824}
SPL {X  -154.891, Y  +711.608, Z    +0.000, E1   -54.831, E3 +23767.211}
SPL {X  -152.273, Y  +720.623, Z    +0.000, E1   -54.369, E3 +23782.949}
SPL {X  -149.300, Y  +729.027, Z    +0.000, E1   -53.836, E3 +23798.085}
SPL {X  -146.549, Y  +735.713, Z    +0.000, E1   -53.293, E3 +23810.499}
SPL {X  -144.128, Y  +740.978, Z    +0.000, E1   -52.835, E3 +23820.462}
SPL {X  -141.140, Y  +746.862, Z    +0.000, E1   -52.272, E3 +23831.750}
SPL {X  -128.473, Y  +766.865, Z    +0.000, E1   -45.208, E3 +23925.959}
ENDSPLINE

SPLINE
SPL {X  -149.609, Y  +728.220, Z    +0.000, E1   -30.103, E3 +24011.652}
SPL {X  -157.346, Y  +700.520, Z    +0.000, E1   -17.449, E3 +24026.373}
SPL {X  -159.391, Y  +685.442, Z    +0.000, E1    -8.940, E3 +24030.258}
SPL {X  -159.974, Y  +674.384, Z    +0.000, E1    -1.914, E3 +24031.609}
SPL {X  -160.000, Y  +668.854, Z    +0.000, E1    +3.008, E3 +24031.960}
SPL {X  -160.000, Y  +662.175, Z    +0.000, E1   +11.518, E3 +24032.731}
SPL {X  -160.000, Y  +654.447, Z    +0.000, E1   +21.734, E3 +24034.357}
SPL {X  -160.000, Y  +641.600, Z    +0.000, E1   +35.681, E3 +24038.622}
SPL {X  -160.000, Y  +601.361, Z    +0.000, E1   +52.744, E3 +24062.584}
SPL {X  -160.000, Y  +531.662, Z    +0.000, E1   +56.951, E3 +24134.573}
SPL {X  -160.000, Y  +513.172, Z    +0.000, E1   +56.969, E3 +24160.129}
SPL {X  -160.000, Y  +498.160, Z    +0.000, E1   +56.531, E3 +24183.741}
ENDSPLINE

SPLINE
SPL {X  -160.000, Y  +512.094, Z    +0.000, E1   +49.085, E3 +24207.729}
ENDSPLINE

SPLINE
SPL {X  -160.000, Y  +491.347, Z    +0.000, E1   +50.960, E3 +24233.396}
SPL {X  -160.000, Y  +470.538, Z    +0.000, E1   +52.629, E3 +24258.082}
SPL {X  -160.000, Y  +453.213, Z    +0.000, E1   +53.894, E3 +24277.520}
SPL {X  -160.000, Y  +440.734, Z    +0.000, E1   +54.729, E3 +24291.302}
SPL {X  -160.000, Y  +423.596, Z    +0.000, E1   +55.911, E3 +24309.194}
SPL {X  -160.000, Y  +408.178, Z    +0.000, E1   +56.432, E3 +24327.655}
SPL {X  -160.000, Y  +395.668, Z    +0.000, E1   +56.446, E3 +24345.270}
SPL {X  -159.894, Y  +382.991, Z    +0.000, E1   +56.419, E3 +24363.268}
SPL {X  -159.213, Y  +372.948, Z    +0.000, E1   +56.290, E3 +24378.163}
SPL {X  -158.141, Y  +364.480, Z    +0.000, E1   +56.110, E3 +24391.237}
SPL {X  -156.499, Y  +355.511, Z    +0.000, E1   +55.854, E3 +24405.553}
SPL {X  -154.489, Y  +347.168, Z    +0.000, E1   +55.487, E3 +24419.428}
SPL {X  -152.108, Y  +339.170, Z    +0.000, E1   +55.085, E3 +24433.117}
SPL {X  -149.149, Y  +330.880, Z    +0.000, E1   +54.560, E3 +24447.753}
SPL {X  -146.188, Y  +323.769, Z    +0.000, E1   +53.991, E3 +24460.709}
SPL {X  -143.516, Y  +318.068, Z    +0.000, E1   +53.476, E3 +24471.309}
SPL {X  -140.415, Y  +312.095, Z    +0.000, E1   +52.896, E3 +24482.576}
SPL {X  -128.706, Y  +293.749, Z    +0.000, E1   +44.636, E3 +24584.637}
ENDSPLINE

SPLINE
SPL {X  -149.341, Y  +331.377, Z    +0.000, E1   +30.257, E3 +24664.512}
SPL {X  -155.855, Y  +352.616, Z    +0.000, E1   +20.935, E3 +24676.625}
SPL {X  -158.820, Y  +369.405, Z    +0.000, E1   +11.982, E3 +24682.029}
SPL {X  -159.764, Y  +380.110, Z    +0.000, E1    +5.506, E3 +24683.896}
SPL {X  -159.978, Y  +386.129, Z    +0.000, E1    +1.351, E3 +24684.478}
SPL {X  -160.000, Y  +390.626, Z    +0.000, E1    -2.404, E3 +24684.742}
SPL {X  -160.000, Y  +397.252, Z    +0.000, E1   -10.844, E3 +24685.443}
SPL {X  -160.000, Y  +404.580, Z    +0.000, E1   -20.626, E3 +24686.868}
SPL {X  -160.000, Y  +414.518, Z    +0.000, E1   -32.156, E3 +24689.959}
SPL {X  -160.000, Y  +450.190, Z    +0.000, E1   -50.789, E3 +24710.045}
SPL {X  -160.000, Y  +522.988, Z    +0.000, E1   -55.744, E3 +24788.379}
SPL {X  -160.000, Y  +538.972, Z    +0.000, E1   -55.709, E3 +24811.611}
SPL {X  -160.000, Y  +554.704, Z    +0.000, E1   -55.732, E3 +24834.378}
SPL {X  -160.000, Y  +570.552, Z    +0.000, E1   -55.716, E3 +24857.392}
SPL {X  -160.000, Y  +586.464, Z    +0.000, E1   -55.733, E3 +24880.438}
SPL {X  -160.000, Y  +602.947, Z    +0.000, E1   -55.730, E3 +24904.334}
SPL {X  -160.000, Y  +618.907, Z    +0.000, E1   -55.724, E3 +24927.472}
SPL {X  -160.000, Y  +633.674, Z    +0.000, E1   -55.717, E3 +24948.892}
SPL {X  -160.000, Y  +646.135, Z    +0.000, E1   -55.674, E3 +24967.033}
SPL {X  -160.000, Y  +658.587, Z    +0.000, E1   -55.708, E3 +24985.029}
SPL {X  -160.000, Y  +671.750, Z    +0.000, E1   -55.695, E3 +25004.113}
SPL {X  -159.611, Y  +682.650, Z    +0.000, E1   -55.614, E3 +25020.351}
SPL {X  -158.677, Y  +692.037, Z    +0.000, E1   -55.461, E3 +25034.934}
SPL {X  -157.091, Y  +701.873, Z    +0.000, E1   -55.210, E3 +25050.821}
SPL {X  -154.891, Y  +711.608, Z    +0.000, E1   -54.831, E3 +25067.207}
SPL {X  -152.273, Y  +720.623, Z    +0.000, E1   -54.369, E3 +25082.945}
SPL {X  -149.300, Y  +729.027, Z    +0.000, E1   -53.836, E3 +25098.081}
SPL {X  -146.549, Y  +735.713, Z    +0.000, E1   -53.293, E3 +25110.496}
SPL {X  -144.128, Y  +740.978, Z    +0.000, E1   -52.835, E3 +25120.458}
SPL {X  -141.140, Y  +746.862, Z    +0.000, E1   -52.272, E3 +25131.746}
SPL {X  -128.473, Y  +766.865, Z    +0.000, E1   -45.208, E3 +25225.955}
ENDSPLINE

SPLINE
SPL {X  -149.609, Y  +728.220, Z    +0.000, E1   -30.103, E3 +25311.648}
SPL {X  -157.346, Y  +700.520, Z    +0.000, E1   -17.449, E3 +25326.369}
SPL {X  -159.391, Y  +685.442, Z    +0.000, E1    -8.940, E3 +25330.254}
SPL {X  -159.974, Y  +674.384, Z    +0.000, E1    -1.914, E3 +25331.606}
SPL {X  -160.000, Y  +668.854, Z    +0.000, E1    +3.008, E3 +25331.957}
SPL {X  -160.000, Y  +662.175, Z    +0.000, E1   +11.518, E3 +25332.728}
SPL {X  -160.000, Y  +654.447, Z    +0.000, E1   +21.734, E3 +25334.353}
SPL {X  -160.000, Y  +641.600, Z    +0.000, E1   +35.681, E3 +25338.618}
SPL {X  -160.000, Y  +601.361, Z    +0.000, E1   +52.744, E3 +25362.580}
SPL {X  -160.000, Y  +531.662, Z    +0.000, E1   +56.951, E3 +25434.569}
SPL {X  -160.000, Y  +513.172, Z    +0.000, E1   +56.969, E3 +25460.125}
SPL {X  -160.000, Y  +498.160, Z    +0.000, E1   +56.531, E3 +25483.738}
ENDSPLINE

SPLINE
SPL {X  -160.000, Y  +512.094, Z    +0.000, E1   +49.085, E3 +25507.726}
ENDSPLINE

SPLINE
SPL {X  -160.000, Y  +491.347, Z    +0.000, E1   +50.960, E3 +25533.392}
SPL {X  -160.000, Y  +470.538, Z    +0.000, E1   +52.629, E3 +25558.078}
SPL {X  -160.000, Y  +453.213, Z    +0.000, E1   +53.894, E3 +25577.516}
SPL {X  -160.000, Y  +440.734, Z    +0.000, E1   +54.729, E3 +25591.298}
SPL {X  -160.000, Y  +423.596, Z    +0.000, E1   +55.911, E3 +25609.190}
ENDSPLINE

SPLINE
SPL {X  -160.000, Y  +422.668, Z    +0.000, E1   +53.123, E3 +25627.801}
SPL {X  -160.000, Y  +412.343, Z    +0.000, E1   +53.116, E3 +25644.273}
SPL {X  -160.000, Y  +402.505, Z    +0.000, E1   +53.115, E3 +25659.946}
SPL {X  -160.000, Y  +391.565, Z    +0.000, E1   +53.135, E3 +25677.353}
SPL {X  -159.782, Y  +380.451, Z    +0.000, E1   +53.086, E3 +25695.315}
SPL {X  -159.005, Y  +370.988, Z    +0.000, E1   +52.949, E3 +25711.214}
SPL {X  -157.765, Y  +362.152, Z    +0.000, E1   +52.730, E3 +25726.613}
SPL {X  -156.057, Y  +353.496, Z    +0.000, E1   +52.443, E3 +25742.151}
SPL {X  -153.530, Y  +343.760, Z    +0.000, E1   +52.025, E3 +25760.204}
SPL {X  -150.540, Y  +334.599, Z    +0.000, E1   +51.451, E3 +25777.853}
SPL {X  -147.202, Y  +326.099, Z    +0.000, E1   +50.843, E3 +25794.646}
SPL {X  -143.559, Y  +318.154, Z    +0.000, E1   +50.126, E3 +25810.793}
SPL {X  -132.920, Y  +299.736, Z    +0.000, E1   +44.141, E3 +25891.938}
ENDSPLINE

SPLINE
SPL {X  -143.903, Y  +318.857, Z    +0.000, E1   +34.827, E3 +25956.086}
SPL {X  -153.845, Y  +344.850, Z    +0.000, E1   +24.318, E3 +25982.181}
SPL {X  -158.184, Y  +364.762, Z    +0.000, E1   +14.458, E3 +25991.560}
SPL {X  -159.644, Y  +378.137, Z    +0.000, E1    +6.763, E3 +25994.874}
SPL {X  -159.957, Y  +385.097, Z    +0.000, E1    +2.214, E3 +25995.790}
SPL {X  -160.000, Y  +390.467, Z    +0.000, E1    -1.886, E3 +25996.231}
SPL {X  -160.000, Y  +396.882, Z    +0.000, E1    -9.361, E3 +25996.984}
SPL {X  -160.000, Y  +403.298, Z    +0.000, E1   -17.340, E3 +25998.287}
SPL {X  -160.000, Y  +414.216, Z    +0.000, E1   -29.557, E3 +26001.836}
SPL {X  -160.000, Y  +448.199, Z    +0.000, E1   -47.246, E3 +26024.329}
SPL {X  -160.000, Y  +510.996, Z    +0.000, E1   -52.996, E3 +26096.653}
SPL {X  -160.000, Y  +527.680, Z    +0.000, E1   -53.008, E3 +26123.422}
SPL {X  -160.000, Y  +543.568, Z    +0.000, E1   -52.978, E3 +26148.962}
SPL {X  -160.000, Y  +558.178, Z    +0.000, E1   -52.971, E3 +26172.421}
SPL {X  -160.000, Y  +573.149, Z    +0.000, E1   -52.983, E3 +26196.435}
SPL {X  -160.000, Y  +589.074, Z    +0.000, E1   -52.998, E3 +26221.976}
SPL {X  -160.000, Y  +605.389, Z    +0.000, E1   -52.996, E3 +26248.176}
SPL {X  -160.000, Y  +621.194, Z    +0.000, E1   -52.986, E3 +26273.576}
SPL {X  -160.000, Y  +634.261, Z    +0.000, E1   -52.926, E3 +26294.655}
SPL {X  -160.000, Y  +645.165, Z    +0.000, E1   -52.917, E3 +26312.174}
SPL {X  -160.000, Y  +655.362, Z    +0.000, E1   -52.919, E3 +26328.525}
SPL {X  -160.000, Y  +666.642, Z    +0.000, E1   -52.938, E3 +26346.601}
SPL {X  -159.882, Y  +677.646, Z    +0.000, E1   -52.897, E3 +26364.432}
SPL {X  -159.100, Y  +688.445, Z    +0.000, E1   -52.790, E3 +26382.555}
SPL {X  -157.767, Y  +698.140, Z    +0.000, E1   -52.527, E3 +26399.566}
SPL {X  -155.944, Y  +707.296, Z    +0.000, E1   -52.232, E3 +26416.124}
SPL {X  -153.388, Y  +717.020, Z    +0.000, E1   -51.781, E3 +26434.329}
SPL {X  -150.628, Y  +725.455, Z    +0.000, E1   -51.252, E3 +26450.687}
SPL {X  -147.586, Y  +733.294, Z    +0.000, E1   -50.691, E3 +26466.264}
SPL {X  -144.002, Y  +741.239, Z    +0.000, E1   -50.009, E3 +26482.440}
SPL {X  -134.968, Y  +757.427, Z    +0.000, E1   -43.006, E3 +26567.718}
ENDSPLINE

SPLINE
SPL {X  -150.251, Y  +726.498, Z    +0.000, E1   -29.147, E3 +26642.704}
SPL {X  -158.295, Y  +694.796, Z    +0.000, E1   -14.337, E3 +26660.696}
SPL {X  -159.852, Y  +678.369, Z    +0.000, E1    -4.607, E3 +26664.640}
SPL {X  -159.994, Y  +672.856, Z    +0.000, E1    -0.741, E3 +26665.228}
SPL {X  -160.000, Y  +667.974, Z    +0.000, E1    +3.384, E3 +26665.656}
SPL {X  -160.000, Y  +657.936, Z    +0.000, E1   +15.171, E3 +26667.408}
SPL {X  -160.000, Y  +643.339, Z    +0.000, E1   +31.330, E3 +26672.400}
SPL {X  -160.000, Y  +606.884, Z    +0.000, E1   +47.933, E3 +26698.255}
SPL {X  -160.000, Y  +552.863, Z    +0.000, E1   +52.205, E3 +26764.060}
SPL {X  -160.000, Y  +541.250, Z    +0.000, E1   +52.128, E3 +26783.364}
SPL {X  -160.000, Y  +532.225, Z    +0.000, E1   +52.130, E3 +26798.271}
SPL {X  -160.000, Y  +522.908, Z    +0.000, E1   +52.129, E3 +26813.675}
SPL {X  -160.000, Y  +514.018, Z    +0.000, E1   +52.121, E3 +26828.360}
SPL {X  -160.000, Y  +502.148, Z    +0.000, E1   +52.197, E3 +26847.836}
SPL {X  -160.000, Y  +488.825, Z    +0.000, E1   +51.737, E3 +26872.881}
ENDSPLINE

SPLINE
SPL {X  -160.000, Y  +489.568, Z    +0.000, E1   +48.224, E3 +26891.905}
ENDSPLINE

SPLINE
SPL {X  -160.000, Y  +479.301, Z    +0.000, E1   +49.113, E3 +26905.783}
SPL {X  -160.000, Y  +468.407, Z    +0.000, E1   +50.011, E3 +26920.110}
SPL {X  -160.000, Y  +457.258, Z    +0.000, E1   +50.929, E3 +26934.095}
SPL {X  -160.000, Y  +444.555, Z    +0.000, E1   +51.931, E3 +26949.579}
SPL {X  -160.000, Y  +432.374, Z    +0.000, E1   +52.787, E3 +26964.204}
SPL {X  -160.000, Y  +422.570, Z    +0.000, E1   +53.120, E3 +26977.962}
SPL {X  -160.000, Y  +412.343, Z    +0.000, E1   +53.116, E3 +26994.269}
SPL {X  -160.000, Y  +402.505, Z    +0.000, E1   +53.115, E3 +27009.941}
SPL {X  -160.000, Y  +391.565, Z    +0.000, E1   +53.135, E3 +27027.348}
SPL {X  -159.782, Y  +380.451, Z    +0.000, E1   +53.086, E3 +27045.311}
SPL {X  -159.005, Y  +370.988, Z    +0.000, E1   +52.949, E3 +27061.210}
SPL {X  -157.765, Y  +362.152, Z    +0.000, E1   +52.730, E3 +27076.608}
SPL {X  -156.057, Y  +353.496, Z    +0.000, E1   +52.443, E3 +27092.147}
SPL {X  -153.530, Y  +343.760, Z    +0.000, E1   +52.025, E3 +27110.200}
SPL {X  -150.540, Y  +334.599, Z    +0.000, E1   +51.451, E3 +27127.848}
SPL {X  -147.202, Y  +326.099, Z    +0.000, E1   +50.843, E3 +27144.642}
SPL {X  -143.559, Y  +318.154, Z    +0.000, E1   +50.126, E3 +27160.789}
SPL {X  -132.920, Y  +299.736, Z    +0.000, E1   +44.141, E3 +27241.933}
ENDSPLINE

